IF bCalculateEnergySession THEN 
		//Socket 1
		IF FPMode3C2[1].Q OR FPMode3D2[1].Q THEN
			//Reset Counter when a new session is started
			stDataECSOut.arrSocketEnergySession[1] := 0;
				//Copy the Total Counter in kWh when a new session is started
				IF IsFinite(F_LREAL(arrSocketEnergySession[1])) THEN
					arrEnergySession_Cmp[1] := arrSocketEnergySession[1];
				END_IF
		END_IF
			IF (arrEnergySession_Cmp[1] <> arrSocketEnergySession[1] AND IsFinite(F_LREAL(arrSocketEnergySession[1])) AND (arrSocketMode3StateECS[1] = 'C2' OR arrSocketMode3StateECS[1] = 'D2')) THEN
				stDataECSOut.arrSocketEnergySession[1] := stDataECSOut.arrSocketEnergySession[1] + (arrSocketEnergySession[1] - arrEnergySession_Cmp[1]) / 1000;  
					stDataECSOut.arrSocketEnergySession[1] := stDataECSOut.arrSocketEnergySession[1];
						arrEnergySession_Cmp[1] := arrSocketEnergySession[1];		
			END_IF
		//Socket 2
		IF FPMode3C2[2].Q OR FPMode3D2[2].Q THEN
			//Reset Counter when a new session is started
			stDataECSOut.arrSocketEnergySession[2] := 0;
				//Copy the Total Counter in kWh when a new session is started
				IF IsFinite(F_LREAL(arrSocketEnergySession[2])) THEN
					arrEnergySession_Cmp[2] := arrSocketEnergySession[2];
				END_IF
		END_IF
			IF (arrEnergySession_Cmp[2] <> arrSocketEnergySession[2] AND IsFinite(F_LREAL(arrSocketEnergySession[2])) AND (arrSocketMode3StateECS[2] = 'C2' OR arrSocketMode3StateECS[2] = 'D2')) THEN
				stDataECSOut.arrSocketEnergySession[2] := stDataECSOut.arrSocketEnergySession[2] + (arrSocketEnergySession[2] - arrEnergySession_Cmp[2]) / 1000;  
					stDataECSOut.arrSocketEnergySession[2] := stDataECSOut.arrSocketEnergySession[2];
						arrEnergySession_Cmp[2] := arrSocketEnergySession[2];		
			END_IF
		//Socket 3
		IF FPMode3C2[3].Q OR FPMode3D2[3].Q THEN
			//Reset Counter when a new session is started
			stDataECSOut.arrSocketEnergySession[3] := 0;
				//Copy the Total Counter in kWh when a new session is started
				IF IsFinite(F_LREAL(arrSocketEnergySession[3])) THEN
					arrEnergySession_Cmp[3] := arrSocketEnergySession[3];
				END_IF
		END_IF
			IF (arrEnergySession_Cmp[3] <> arrSocketEnergySession[3] AND IsFinite(F_LREAL(arrSocketEnergySession[3])) AND (arrSocketMode3StateECS[3] = 'C2' OR arrSocketMode3StateECS[3] = 'D2')) THEN
				stDataECSOut.arrSocketEnergySession[3] := stDataECSOut.arrSocketEnergySession[3] + (arrSocketEnergySession[3] - arrEnergySession_Cmp[3]) / 1000;  
					stDataECSOut.arrSocketEnergySession[3] := stDataECSOut.arrSocketEnergySession[3];
						arrEnergySession_Cmp[3] := arrSocketEnergySession[3];		
			END_IF
		//Socket 4
		IF FPMode3C2[4].Q OR FPMode3D2[4].Q THEN
			//Reset Counter when a new session is started
			stDataECSOut.arrSocketEnergySession[4] := 0;
				//Copy the Total Counter in kWh when a new session is started
				IF IsFinite(F_LREAL(arrSocketEnergySession[4])) THEN
					arrEnergySession_Cmp[4] := arrSocketEnergySession[4];
				END_IF
		END_IF
			IF (arrEnergySession_Cmp[4] <> arrSocketEnergySession[4] AND IsFinite(F_LREAL(arrSocketEnergySession[4])) AND (arrSocketMode3StateECS[4] = 'C2' OR arrSocketMode3StateECS[4] = 'D2')) THEN
				stDataECSOut.arrSocketEnergySession[4] := stDataECSOut.arrSocketEnergySession[4] + (arrSocketEnergySession[4] - arrEnergySession_Cmp[4]) / 1000;  
					stDataECSOut.arrSocketEnergySession[4] := stDataECSOut.arrSocketEnergySession[4];
						arrEnergySession_Cmp[4] := arrSocketEnergySession[4];		
			END_IF
			
		stDataECSOut.arrSocketEnergySession[1] := LINT_TO_LREAL(LREAL_TO_LINT(stDataECSOut.arrSocketEnergySession[1] * 1000)) / 1000;
		stDataECSOut.arrSocketEnergySession[2] := LINT_TO_LREAL(LREAL_TO_LINT(stDataECSOut.arrSocketEnergySession[2] * 1000)) / 1000;
		stDataECSOut.arrSocketEnergySession[3] := LINT_TO_LREAL(LREAL_TO_LINT(stDataECSOut.arrSocketEnergySession[3] * 1000)) / 1000;
		stDataECSOut.arrSocketEnergySession[4] := LINT_TO_LREAL(LREAL_TO_LINT(stDataECSOut.arrSocketEnergySession[4] * 1000)) / 1000;
			
ELSE
	IF IsFinite(F_LREAL(arrSocketEnergySession[1])) THEN stDataECSOut.arrSocketEnergySession[1] := LINT_TO_LREAL(LREAL_TO_LINT((arrSocketEnergySession[1] / 1000) * 1000)) / 1000; END_IF
		IF IsFinite(F_LREAL(arrSocketEnergySession[2])) THEN stDataECSOut.arrSocketEnergySession[2] := LINT_TO_LREAL(LREAL_TO_LINT((arrSocketEnergySession[2] / 1000) * 1000)) / 1000; END_IF
			IF IsFinite(F_LREAL(arrSocketEnergySession[3])) THEN stDataECSOut.arrSocketEnergySession[3] := LINT_TO_LREAL(LREAL_TO_LINT((arrSocketEnergySession[3] / 1000) * 1000)) / 1000; END_IF
				IF IsFinite(F_LREAL(arrSocketEnergySession[4])) THEN stDataECSOut.arrSocketEnergySession[4] := LINT_TO_LREAL(LREAL_TO_LINT((arrSocketEnergySession[4] / 1000) * 1000)) / 1000; END_IF
END_IF
		
(*---------------------------------------------------------------------------Outputs--------------------------------------------------------------------------------------*)

stDataECSOut.byPriority := stSetupECS.byPriority;
	stDataECSOut.rMaxPower := DINT_TO_REAL(REAL_TO_DINT(stSetupECS.rMaxPower * 100)) / 100;
		stDataECSOut.bSOnEmergPowerOff := stSetupECS.bOnEmergPowerOff;
			stDataECSOut.bSManualyOn := stSetupECS.bManualyOn;
				stDataECSOut.bySManualyTargetPower := stSetupECS.byManualyTargetPower;
					stDataECSOut.bySCSMinPower := stSetupECS.byCSMinPower;

stDataECSOut.bCarConnected := bCarConnected;

//Mode 3 State
//Socket 1
//No Value.
IF arrSocketMode3StateECS[1] = '' OR arrSocketMode3StateECS[1] = 'F' OR NOT bEnable THEN
	stDataECSOut.arrSocketStateECS[1] := 0;
//ECS ready and Free	
ELSIF arrSocketMode3StateECS[1] = 'A' OR arrSocketMode3StateECS[1] = 'E' THEN
	stDataECSOut.arrSocketStateECS[1] := 1;
//Car Connected
ELSIF arrSocketMode3StateECS[1] = 'B1' OR arrSocketMode3StateECS[1] = 'B2' OR arrSocketMode3StateECS[1] = 'C1' OR arrSocketMode3StateECS[1] = 'D1' THEN
	stDataECSOut.arrSocketStateECS[1] := 2;
//Car Charging
ELSIF arrSocketMode3StateECS[1] = 'C2' OR arrSocketMode3StateECS[1] = 'D2' THEN
	stDataECSOut.arrSocketStateECS[1] := 3;
END_IF
//Socket 2
//No Value.
IF arrSocketMode3StateECS[2] = '' OR arrSocketMode3StateECS[2] = 'F' OR NOT bEnable THEN
	stDataECSOut.arrSocketStateECS[2] := 0;
//ECS ready and Free	
ELSIF arrSocketMode3StateECS[2] = 'A' OR arrSocketMode3StateECS[2] = 'E' THEN
	stDataECSOut.arrSocketStateECS[2] := 1;
//Car Connected
ELSIF arrSocketMode3StateECS[2] = 'B1' OR arrSocketMode3StateECS[2] = 'B2' OR arrSocketMode3StateECS[2] = 'C1' OR arrSocketMode3StateECS[2] = 'D1' THEN
	stDataECSOut.arrSocketStateECS[2] := 2;
//Car Charging
ELSIF arrSocketMode3StateECS[2] = 'C2' OR arrSocketMode3StateECS[2] = 'D2' THEN
	stDataECSOut.arrSocketStateECS[2] := 3;
END_IF
//Socket 3
//No Value.
IF arrSocketMode3StateECS[3] = '' OR arrSocketMode3StateECS[3] = 'F' OR NOT bEnable THEN
	stDataECSOut.arrSocketStateECS[3] := 0;
//ECS ready and Free	
ELSIF arrSocketMode3StateECS[3] = 'A' OR arrSocketMode3StateECS[3] = 'E' THEN
	stDataECSOut.arrSocketStateECS[3] := 1;
//Car Connected
ELSIF arrSocketMode3StateECS[3] = 'B1' OR arrSocketMode3StateECS[3] = 'B2' OR arrSocketMode3StateECS[3] = 'C1' OR arrSocketMode3StateECS[3] = 'D1' THEN
	stDataECSOut.arrSocketStateECS[3] := 2;
//Car Charging
ELSIF arrSocketMode3StateECS[3] = 'C2' OR arrSocketMode3StateECS[3] = 'D2' THEN
	stDataECSOut.arrSocketStateECS[3] := 3;
END_IF
//Socket 4
//No Value.
IF arrSocketMode3StateECS[4] = '' OR arrSocketMode3StateECS[4] = 'F' OR NOT bEnable THEN
	stDataECSOut.arrSocketStateECS[4] := 0;
//ECS ready and Free	
ELSIF arrSocketMode3StateECS[4] = 'A' OR arrSocketMode3StateECS[4] = 'E' THEN
	stDataECSOut.arrSocketStateECS[4] := 1;
//Car Connected
ELSIF arrSocketMode3StateECS[4] = 'B1' OR arrSocketMode3StateECS[4] = 'B2' OR arrSocketMode3StateECS[4] = 'C1' OR arrSocketMode3StateECS[4] = 'D1' THEN
	stDataECSOut.arrSocketStateECS[4] := 2;
//Car Charging
ELSIF arrSocketMode3StateECS[4] = 'C2' OR arrSocketMode3StateECS[4] = 'D2' THEN
	stDataECSOut.arrSocketStateECS[4] := 3;
END_IF
	
IF bEnable THEN
	stDataECSOut.arrSocketSOCCar[1] := arrSOCCar[1];
	stDataECSOut.arrSocketSOCCar[2] := arrSOCCar[2];
	stDataECSOut.arrSocketSOCCar[3] := arrSOCCar[3];
	stDataECSOut.arrSocketSOCCar[4] := arrSOCCar[4];
		stDataECSOut.arrChargingTimeInMin[1] := DINT_TO_REAL(REAL_TO_DINT(arrSocketChargingTimeInput[1] * 100)) / 100;
		stDataECSOut.arrChargingTimeInMin[2] := DINT_TO_REAL(REAL_TO_DINT(arrSocketChargingTimeInput[2] * 100)) / 100;
		stDataECSOut.arrChargingTimeInMin[3] := DINT_TO_REAL(REAL_TO_DINT(arrSocketChargingTimeInput[3] * 100)) / 100;
		stDataECSOut.arrChargingTimeInMin[4] := DINT_TO_REAL(REAL_TO_DINT(arrSocketChargingTimeInput[4] * 100)) / 100;
ELSE
	stDataECSOut.arrSocketSOCCar[1] := 0;
	stDataECSOut.arrSocketSOCCar[2] := 0;
	stDataECSOut.arrSocketSOCCar[3] := 0;
	stDataECSOut.arrSocketSOCCar[4] := 0;
		stDataECSOut.arrChargingTimeInMin[1] := 0;
		stDataECSOut.arrChargingTimeInMin[2] := 0;
		stDataECSOut.arrChargingTimeInMin[3] := 0;
		stDataECSOut.arrChargingTimeInMin[4] := 0;
END_IF

timDelayOutputs(IN:= bWriteWithDelay AND bEnable AND NOT timDelayOutputs.Q, PT:= tTimDelayOutput, Q=> , ET=> );
	FPEnable(CLK:= bEnable, Q=> );
		FNEnable(CLK:= bEnable, Q=> );
		
//Write with Delay or without
IF (bWriteWithDelay AND (timDelayOutputs.Q OR FPEnable.Q OR FNEnable.Q)) OR NOT bWriteWithDelay THEN
	stDataECSOutDelay := stDataECSOut;
END_IF

END_FUNCTION_BLOCK

// ---- Energy/FBs Internal/Electric Heating Element/FB_ElectricHeatingElement.TcPOU
{attribute 'conditionalshow'}
FUNCTION_BLOCK FB_ElectricHeatingElement
VAR_INPUT
	{attribute 'hide'}
	bEnable								: BOOL;									//Enable the Fuctionblock and his logic
	{attribute 'hide'}
	bError								: BOOL;									//Error Input electric heating element
	{attribute 'hide'}
	bWarning							: BOOL;									//Warning Input electric heating element
	{attribute 'hide'}
	bIsStepSwitched						: BOOL;									//Heating element is step switched or not
	{attribute 'hide'}
	bEPOIsActive						: BOOL;									//Emergency power operation is active
	{attribute 'hide'}
	bExternalLock						: BOOL;									//External lock (All functions are locked)
	{attribute 'hide'}
	bWriteWithDelay						: BOOL;									//Write with Delay the Data to the output (Not al Output Data is writen with Delay)
	{attribute 'hide'}
	bTimeDissableFunctions				: BOOL;									//True when we have longer Time no conncection to the Backend System. We need this Information to switch on the Heating Element for the Legionella Prtection
	{attribute 'hide'}
	iErrorCode							: INT;									//Error Code from external EHE
	{attribute 'hide'}
	iWarningCode						: INT;									//Warning Code from external EHE
	{attribute 'hide'}
	diNumberOfEHE						: DINT;									//Number of Electric Heating Element what is calculatet by a external function
	{attribute 'hide'}
	dwBatterySOC						: DWORD;								//Actual Battery SOC in %
	{attribute 'hide'}
	lrSizeGridConnection				: LREAL;								//Max size from the grid connection in kW
	{attribute 'hide'}
	lrGridPower							: LREAL;								//Actual Grid power in kW
	{attribute 'hide'}
	lrTotalCounterEnergy_Consumption	: LREAL;								//Total Counter for Energy consumption with unit Wh
	{attribute 'hide'}
	lrTotalCounterEnergy_Production		: LREAL;								//Total Counter for Energy production with unit Wh
	{attribute 'hide'}
	lrCounterEnergyT1_Consumption		: LREAL;								//Total counter for energy Tariff 1 consumption with unit Wh
	{attribute 'hide'}
	lrCounterEnergyT2_Consumption		: LREAL;								//Total counter for energy Tariff 2 consumption with unit Wh
	{attribute 'hide'}
	lrCounterEnergyT1_Production		: LREAL;								//Total counter for energy Tariff 1 production with unit Wh
	{attribute 'hide'}
	lrCounterEnergyT2_Production		: LREAL;								//Total counter for energy Tariff 2 production with unit Wh
	{attribute 'hide'}
	lrPowerEHE							: LREAL;								//Input Value from the power of the electro heating element with unit W
	{attribute 'hide'}
	arrTargetPower						: ARRAY[1..10] OF REAL;					//Target power from 0% to +100% for each step (0% to 100%) 
	{attribute 'hide'}
	rTemperatureInBoiler				: REAL;									//Temperature in the boiler which is heated with the heating element
	{attribute 'hide'}
	tTimDelayOutput						: TIME := T#5S;							//Delay Time to write some Data to the Output
	{attribute 'hide'}
	stSystemTime						: ST_Systemtime;						//Local System Time
	{attribute 'hide'}
	stSetupEHE							: ST_Setup_EHE;							//Setup electric heating element
END_VAR
VAR_OUTPUT
	{attribute 'hide'}
	stDataEHEOut						: ST_EHE_Output;						//Electric heating element output data
	{attribute 'hide'}
	stDataEHEOutDelay					: ST_EHE_Output;						//Electric heating element output data with delay
END_VAR
VAR
	{attribute 'hide'}
	fbPD1								: FB_PersistentData_Number;				//Function to save persistent data
	{attribute 'hide'}
	fbPD2								: FB_PersistentData_Number;				//Function to save persistent data
	{attribute 'hide'}
	FPTimeEnable						: R_TRIG;								//Internal positive edge
	{attribute 'hide'}
	FPTimeDisable						: R_TRIG;								//Internal positive edge
	{attribute 'hide'}
	FPWeekProgram						: R_TRIG;								//Internal positive edge
	{attribute 'hide'}
	FPRSWeekProgram						: R_TRIG;								//Internal positive edge
	{attribute 'hide'}
	FPEnable							: R_TRIG;								//Internal positive Edge
	{attribute 'hide'}
	FNEnable							: F_TRIG;								//Internal negative Edge
	{attribute 'hide'}
	timError							: TOF;									//Timer to set the error
	{attribute 'hide'}
	timWeekProgram						: TON;									//Timer for the week program (legionella protection)
	{attribute 'hide'}
	timDelayOutputs						: TON;									//Timer to send Data with Delay to the outputs
	{attribute 'hide'}
	timStep5							: TON;									//Timer what show when the state machine is to long in step 5. (The heating element not can heat the boiler at the Temperature what we need for the weekprogram)
	{attribute 'hide'}
	timStep6IsActive					: TON;									//Timer what is active when Step 6 in the State Machine is active
	{attribute 'hide'}
	timOnDelayStep6						: TON;									//Delay to switch on the EHE in Step 6
	{attribute 'hide'}
	timOffDelayStep6					: TON;									//Delay to switch off the EHE in Step 6
	{attribute 'hide'}
	timSOCOff							: TON;									//Timer to dissable the Device when the SOC from the Battery is under the Setpoint
	{attribute 'hide'}
	bTimeIsEnabled						: BOOL;									//Enable time controll
	{attribute 'hide'}
	byLPLimitsPw						: BYTE;									//Loop to check limits for target and max power
	{attribute 'hide'}
	byLPNumberOfSteps					: BYTE;									//Loop to ckeck to number of steps for step switching
	{attribute 'hide'}
	byLPMaxPowerOutput					: BYTE;									//Loop to ckeck the max power befor write to the output
	{attribute 'hide'}
	byLPSumPwOfSteps					: BYTE;									//Loop to calculate the complete power of all steps
	{attribute 'hide'}
	byLPPercentPwOfSteps				: BYTE;									//Loop to calculate the complete power in percent of all steps
	{attribute 'hide'}
	byLPMaxReached						: BYTE;									//Loop to check if for some step the target power is >= 100 or < Constants.byTargetOffPowerOnOffDevices
	{attribute 'hide'}
	iStateIntStep6						: INT;									//Internal Statmachine in Step 6
	{attribute 'hide'}
	uiState								: UINT;									//State Maschine
	{attribute 'hide'}
	uiHysteresisOnStep3					: UINT;									//Hysteresis to switch on or off the heating elemtn in step 3 (Surplus mode and max temperature)
	{attribute 'hide'}
	uiWeekProgramTemp					: UINT;									//Temperature, what is needed for the legionella protection
	{attribute 'hide'}
	rSumSteps							: REAL;									//Sum from all steps 
	{attribute 'hide'}
	arrMaxPower							: ARRAY[1..10] OF REAL; 				//Maximum power of the load in kW (Per stage) (If no stage or only On Off then max power in array[1])	
	{attribute 'hide'}
	arrPercentValueSteps				: ARRAY[1..10] OF REAL;					//Percent Value from each step
	{attribute 'hide'}
	arrMaxReached						: ARRAY[1..10] OF BOOL;					//Array from each step what goes to true when the power is >= 100%
END_VAR
VAR PERSISTENT
	{attribute 'conditionalshow'}
	bWeekProgramEnable					: BOOL;									//Enable the Week programm for one time
	{attribute 'conditionalshow'}
	byCounterDays						: BYTE;									//Counter that counts the days how long has not reached the maximum temperature
END_VAR

//Creator : Kai Ebensperger
//Company : Lynus AG
//Date : 19.05.2021
//Version : 1.0.0.0

//General description:
//This function block implements an electric heating element. It can be used for one adjustable step-switched, one adjustable stepless and one ON/OFF heating element.
//The function block can be switched manually and also contoll based.
//The output bOutputEHEOnOff is set at 100% power input. If the power input is < Constants.byTargetOffPowerOnOffDevices, the output is reset (hysteresis to prevent toggling).
//This output is used for electrical heating elements which cannot be controlled. So only have an on / off function. 
//The output bOutputEHE is set as soon as the power input is greater than or equal to 1%. This output is used for the control of the controllable heating elements. 
//If the temperature falls below the minimum temperature (uiTargetTempOn), the heating element is heated up until the target temperature (uiTargetTempOff) is reached. If time-controlled, this only takes place in the respectively enabled time.
//If a battery cabinet is in emergency power mode at this time, the current SOC must also be above the SOC Off value so that the heating element switches on. This prevents the battery from being discharged.
//IMPORTANT : When controlling the electric heating element, it is important that if it has an integrated mechanical thermostat, this value is set as high as the minimum max. temperature (uiTargetTempMax) set on the PLC. !!Min 65°C!!
//----------------------------------------
//Adjustable stage-switched heating element:
//With the controllable stage-switched heating element, each stage can be given a separate power setting. Each stage can be viewed internally similar to a heating element that can only ON/OFF.
//If >= 100% power output per stage, the percentage value of the respective stage is passed on to the power output (rTargetPowerEHE) or added to it. 
//If the level becomes < Constants.byTargetOffPowerOnOffDevices again, the percentage value is removed from the output again.
//----------------------------------------
//Adjustable stepless heating element:
//In the case of the controllable stepless heating element, the power setting is given linearly to the power setting output (rTargetPowerEHE). 
//The maximum power (arrMaxPowerEHE) must therefore only be entered in the first array field. 
//----------------------------------------
//On-off heating elemet
//Works in the same style like the stepless heating element. But here we use only the output bOutputEHEOnOff to switch on and off the heating element. The rTargetPowerEHE we didn't need here. 
//----------------------------------------
//Timefunctions: 
//If the time function has been selected, the heating element is only controlled if the uiTargetTempOn is undershot between the set time period.
//Is usefully if you have 2 differen current tariffs
//----------------------------------------
//Legionella protection: 
//If the Legionella protection has not been deactivated (bDisableLegionellaProtection), the heating element runs the maximum temperature once every 7 days (if the maximum temperature > 60°C), 
//or 60°C (if maximum temperature < 60°C). If within the 7 days the heating element has already reached the maximum temperature once, the counter, which counts the days will be reset.
//In emergency power mode, the program is only executed if the battery charge level allows it.
//When the Connection to the Backend is lost, then every 5 days the Heating Elemet switch on for 9 hours (In the 9 hours the temperature for legionella protection should be reached)
//----------------------------------------
//On Emergency power operation off
//If the lock for emergency power operation (bOnEmergPowerOff) has been selected for the electric heating element, it will not be switched on in emergency power operation. However, it can be overridden manually.
//----------------------------------------
//External look:
//The FB also has an external inhibit signal which switches off all functions as long as this signal is active.

(*---------------------------------------------------------------Check the limits of the inputs-------------------------------------------------------------------------------*)
dwBatterySOC := LIMIT(0, dwBatterySOC, 100);
	stSetupEHE.byManualyTargetPower := LIMIT(0, stSetupEHE.byManualyTargetPower, 100);
		rTemperatureInBoiler := LIMIT(-30, rTemperatureInBoiler, 120); 
			stSetupEHE.byHourOn := LIMIT(0, stSetupEHE.byHourOn, 23);
				stSetupEHE.byHourOff := LIMIT(0, stSetupEHE.byHourOff, 23);
					stSetupEHE.byMinutesOn := LIMIT(0, stSetupEHE.byMinutesOn, 59);
						stSetupEHE.byMinutesOff := LIMIT(0, stSetupEHE.byMinutesOff, 59);
						
IF IsFinite(F_LREAL(lrTotalCounterEnergy_Consumption)) THEN lrTotalCounterEnergy_Consumption := LIMIT(0,lrTotalCounterEnergy_Consumption,999999999999999); END_IF
	IF IsFinite(F_LREAL(lrTotalCounterEnergy_Production)) THEN lrTotalCounterEnergy_Production := LIMIT(0,lrTotalCounterEnergy_Production,999999999999999); END_IF
		IF IsFinite(F_LREAL(lrCounterEnergyT1_Consumption)) THEN lrCounterEnergyT1_Consumption := LIMIT(0,lrCounterEnergyT1_Consumption,999999999999999); END_IF
			IF IsFinite(F_LREAL(lrCounterEnergyT2_Consumption)) THEN lrCounterEnergyT2_Consumption := LIMIT(0,lrCounterEnergyT2_Consumption,999999999999999); END_IF
				IF IsFinite(F_LREAL(lrCounterEnergyT1_Production)) THEN lrCounterEnergyT1_Production := LIMIT(0,lrCounterEnergyT1_Production,999999999999999); END_IF
					IF IsFinite(F_LREAL(lrCounterEnergyT2_Production)) THEN lrCounterEnergyT2_Production := LIMIT(0,lrCounterEnergyT2_Production,999999999999999); END_IF
						lrPowerEHE := LIMIT(-999999999999999,lrPowerEHE,999999999999999);

//If a maximum power has not been entered everywhere, use the next higher power (only for step-switched). 
IF bIsStepSwitched AND stSetupEHE.rMaxPower1 <= 0 AND stSetupEHE.rMaxPower2 > 0 THEN 
	stSetupEHE.rMaxPower1 := stSetupEHE.rMaxPower2; 
END_IF
	IF bIsStepSwitched AND stSetupEHE.rMaxPower2 <= 0 AND stSetupEHE.rMaxPower3 > 0 THEN 
		stSetupEHE.rMaxPower2 := stSetupEHE.rMaxPower3;
	END_IF
IF bIsStepSwitched AND stSetupEHE.rMaxPower3 <= 0 AND stSetupEHE.rMaxPower4 > 0 THEN 
	stSetupEHE.rMaxPower3 := stSetupEHE.rMaxPower4; 
END_IF
	IF bIsStepSwitched AND stSetupEHE.rMaxPower4 <= 0 AND stSetupEHE.rMaxPower5 > 0 THEN 
		stSetupEHE.rMaxPower4 := stSetupEHE.rMaxPower5; 
	END_IF
IF bIsStepSwitched AND stSetupEHE.rMaxPower5 <= 0 AND stSetupEHE.rMaxPower6 > 0 THEN 
	stSetupEHE.rMaxPower5 := stSetupEHE.rMaxPower6; 
END_IF
	IF bIsStepSwitched AND stSetupEHE.rMaxPower6 <= 0 AND stSetupEHE.rMaxPower7 > 0 THEN 
		stSetupEHE.rMaxPower6 := stSetupEHE.rMaxPower7; 
	END_IF
IF bIsStepSwitched AND stSetupEHE.rMaxPower7 <= 0 AND stSetupEHE.rMaxPower8 > 0 THEN 
	stSetupEHE.rMaxPower7 := stSetupEHE.rMaxPower8; 
END_IF
	IF bIsStepSwitched AND stSetupEHE.rMaxPower8 <= 0 AND stSetupEHE.rMaxPower9 > 0 THEN 
		stSetupEHE.rMaxPower8 := stSetupEHE.rMaxPower9; 
	END_IF
IF bIsStepSwitched AND stSetupEHE.rMaxPower9 <= 0 AND stSetupEHE.rMaxPower10 > 0 THEN 
	stSetupEHE.rMaxPower9 := stSetupEHE.rMaxPower10; 
END_IF						

//Check limits for target power and maximum power						
FOR byLPLimitsPw := 1 TO 10 BY 1 DO
	arrTargetPower[byLPLimitsPw] := LIMIT(0, arrTargetPower[byLPLimitsPw], 100);
END_FOR
	stSetupEHE.rMaxPower1 := LIMIT(0,stSetupEHE.rMaxPower1,500);
		stSetupEHE.rMaxPower2 := LIMIT(0,stSetupEHE.rMaxPower2,500);
			stSetupEHE.rMaxPower3 := LIMIT(0,stSetupEHE.rMaxPower3,500);
				stSetupEHE.rMaxPower4 := LIMIT(0,stSetupEHE.rMaxPower4,500);
					stSetupEHE.rMaxPower5 := LIMIT(0,stSetupEHE.rMaxPower5,500);
						stSetupEHE.rMaxPower6 := LIMIT(0,stSetupEHE.rMaxPower6,500);
							stSetupEHE.rMaxPower7 := LIMIT(0,stSetupEHE.rMaxPower7,500);
								stSetupEHE.rMaxPower8 := LIMIT(0,stSetupEHE.rMaxPower8,500);
									stSetupEHE.rMaxPower9 := LIMIT(0,stSetupEHE.rMaxPower9,500);
										stSetupEHE.rMaxPower10 := LIMIT(0,stSetupEHE.rMaxPower10,500);

//Copy the max input power in the internal array to calculate the steps
arrMaxPower[1] := stSetupEHE.rMaxPower1;
	arrMaxPower[2] := stSetupEHE.rMaxPower2;
		arrMaxPower[3] := stSetupEHE.rMaxPower3;
			arrMaxPower[4] := stSetupEHE.rMaxPower4;
				arrMaxPower[5] := stSetupEHE.rMaxPower5;
					arrMaxPower[6] := stSetupEHE.rMaxPower6;
						arrMaxPower[7] := stSetupEHE.rMaxPower7;
							arrMaxPower[8] := stSetupEHE.rMaxPower8;
								arrMaxPower[9] := stSetupEHE.rMaxPower9;
									arrMaxPower[10] := stSetupEHE.rMaxPower10;

//Check that Disable SOC is bigger then Enable SOC	
IF stSetupEHE.byDisableSOC > stSetupEHE.byEnableSOC THEN 
	stSetupEHE.byEnableSOC := stSetupEHE.byDisableSOC + 1; 
END_IF
	stSetupEHE.byDisableSOC := LIMIT(0, stSetupEHE.byDisableSOC, 100);
		stSetupEHE.byEnableSOC := LIMIT(1, stSetupEHE.byEnableSOC, 100);

//Check that On temperature is bigger than off temperatur	
IF stSetupEHE.uiTargetTempOn > stSetupEHE.uiTargetTempOff THEN 
	stSetupEHE.uiTargetTempOff := stSetupEHE.uiTargetTempOn + 1; 
END_IF
	//Check that max temperature is bigger than on temperatur
	IF stSetupEHE.uiTargetTempOn > stSetupEHE.uiTargetTempMax THEN 
		stSetupEHE.uiTargetTempMax := stSetupEHE.uiTargetTempOn + 1; 
	END_IF
		//Check that max temperature is bigger than off temperatur
		IF stSetupEHE.uiTargetTempOff > stSetupEHE.uiTargetTempMax THEN 
			stSetupEHE.uiTargetTempMax := stSetupEHE.uiTargetTempOff + 1; 
		END_IF  
			stSetupEHE.uiTargetTempOn := LIMIT(0, stSetupEHE.uiTargetTempOn, 120);
				stSetupEHE.uiTargetTempOff := LIMIT(0, stSetupEHE.uiTargetTempOff, 120);
					stSetupEHE.uiTargetTempMax := LIMIT(0, stSetupEHE.uiTargetTempMax, 120);

//Calculate the hysteresis
IF stSetupEHE.uiTargetTempMax >= 2 THEN
	uiHysteresisOnStep3 := 1;
ELSE
	uiHysteresisOnStep3 := 0;
END_IF		

//Check number of steps
stDataEHEOut.byNumberOfSteps := 0;
	FOR byLPNumberOfSteps := 1 TO 10 BY 1 DO
		IF arrMaxPower[byLPNumberOfSteps] > 0 THEN stDataEHEOut.byNumberOfSteps := stDataEHEOut.byNumberOfSteps + 1; END_IF
	END_FOR

//Round the output power
FOR byLPMaxPowerOutput := 1 TO 10 BY 1 DO
	stDataEHEOut.arrMaxPower[byLPMaxPowerOutput] := DINT_TO_REAL(REAL_TO_DINT(arrMaxPower[byLPMaxPowerOutput] * 100)) / 100;
END_FOR	
		
(*---------------------------------------------------------------------------Enable----------------------------------------------------------------------------------*)
stDataEHEOut.bEnabled := bEnable;

(*-----------------------------------------------------------------------------Error and Warning----------------------------------------------------------------------------*)
timError(IN:= bError, PT:= T#5S, Q=> , ET=> );

stDataEHEOut.byErrorWarning := 0;
	IF bWarning OR timStep5.Q THEN stDataEHEOut.byErrorWarning := 1; END_IF 	
	IF timError.Q THEN stDataEHEOut.byErrorWarning := 2; END_IF

//Messages and Error Codes
IF stSetupEHE.bDisableLegionellaPr THEN stDataEHEOut.eMessage := E_Message_EHE.eLegionellaProtectionDisabledFromUser;
ELSIF timStep5.Q THEN stDataEHEOut.eMessage := E_Message_EHE.eEHEDontReachedTheSetTemp;
ELSIF bExternalLock THEN stDataEHEOut.eMessage := E_Message_EHE.eExternalLockActive;
ELSIF stDataEHEOut.byErrorWarning = 1 AND iWarningCode = 0 THEN stDataEHEOut.eMessage := E_Message_EHE.eNoConnectionToBackend;
ELSIF stDataEHEOut.byErrorWarning = 2 AND iErrorCode = 0 THEN stDataEHEOut.eMessage := E_Message_EHE.eErrorEHE;
ELSIF stDataEHEOut.byErrorWarning = 2 AND iErrorCode = 1 THEN stDataEHEOut.eMessage := E_Message_EHE.eTooMuchEHE;
ELSIF stDataEHEOut.byErrorWarning = 2 AND iErrorCode = 2 THEN stDataEHEOut.eMessage := E_Message_EHE.eTempSensorInBufferError;
ELSIF stDataEHEOut.byErrorWarning = 2 AND iErrorCode = 3 THEN stDataEHEOut.eMessage := E_Message_EHE.eWindowsSystemTimeError;	
ELSE stDataEHEOut.eMessage := E_Message_EHE.eNoMessage; 
END_IF
	
(*----------------------------------------------------------------------------Logic Part------------------------------------------------------------------------------------*)

//Timer for SOC dissabling
timSOCOff(IN:= dwBatterySOC <= stSetupEHE.byDisableSOC, PT:= T#30S, Q=> , ET=> );

//Switch heating element depending on temperature (without power setting, without control via time)
IF bEnable AND NOT bWeekProgramEnable AND NOT bExternalLock AND stDataEHEOut.byErrorWarning <> 2 AND 
 rTemperatureInBoiler < stSetupEHE.uiTargetTempOn AND NOT stSetupEHE.bTimeEnabled THEN 
	uiState := 1; 
END_IF

//Switch heating element depending on temperature (without power setting, with control via time)
IF bEnable AND NOT bWeekProgramEnable AND NOT bExternalLock AND stDataEHEOut.byErrorWarning <> 2 AND 
 rTemperatureInBoiler < stSetupEHE.uiTargetTempOn AND stSetupEHE.bTimeEnabled THEN 
	uiState := 2; 
END_IF

//Switch heating element with power preset (surplus)
IF bEnable AND NOT bWeekProgramEnable AND NOT bExternalLock AND stDataEHEOut.byErrorWarning <> 2 AND 
 (arrTargetPower[1] > 0 OR arrTargetPower[2] > 0 OR arrTargetPower[3] > 0 OR arrTargetPower[4] > 0 OR arrTargetPower[5] > 0 OR
 	arrTargetPower[6] > 0 OR arrTargetPower[7] > 0 OR arrTargetPower[8] > 0 OR arrTargetPower[9] > 0 OR arrTargetPower[10] > 0) THEN 
		uiState := 3; 
END_IF

//Switch heating element manually
IF bEnable AND NOT bWeekProgramEnable AND NOT bExternalLock AND stDataEHEOut.byErrorWarning <> 2 AND stSetupEHE.bManualyOn THEN 
	uiState := 4; 
END_IF 

//Legionella protection
IF NOT stSetupEHE.bDisableLegionellaPr THEN
	//Determine the temperature to be approached
	IF stSetupEHE.uiTargetTempMax > 60 THEN
		uiWeekProgramTemp := stSetupEHE.uiTargetTempMax;
	ELSE
		uiWeekProgramTemp := 60;
	END_IF
	
	//Timer and counter for days
	timWeekProgram(IN:= NOT timWeekProgram.Q AND bEnable AND uiState <> 5, PT:=T#24H , Q=> , ET=> );
		FPWeekProgram(CLK:= timWeekProgram.Q, Q=> );
			IF FPWeekProgram.Q THEN 
				byCounterDays := byCounterDays + 1; 
			END_IF
	
	//Reset the counter for the days
	FPRSWeekProgram(CLK:= rTemperatureInBoiler >= uiWeekProgramTemp, Q=> );		
		IF (byCounterDays >= 7 AND rTemperatureInBoiler >= uiWeekProgramTemp) OR FPRSWeekProgram.Q THEN 
			byCounterDays := 0; 
		END_IF
	
	IF byCounterDays >= 7 THEN 
		bWeekProgramEnable := TRUE;
	END_IF 
	
	IF bWeekProgramEnable THEN 
		uiState := 5; 
	END_IF
END_IF

//Timer, when the Weekprogram take to long time and dont reached the Week programm temperature
IF uiState = 5 THEN timStep5.IN := TRUE; ELSE timStep5.IN := FALSE; END_IF
	timStep5(IN:= , PT:= T#12H, Q=> , ET=> );

//Heating Element in Init step (Reset-Off)
IF NOT bEnable OR
	(uiState <> 5 AND (stDataEHEOut.byErrorWarning = 2 OR bExternalLock)) THEN
		uiState := 0;
END_IF

//Activeate the Legionella Protection when the Function is dissabled why we have no connection to the Backend Service
IF NOT bEnable AND bTimeDissableFunctions AND NOT stSetupEHE.bDisableLegionellaPr THEN uiState := 6; END_IF

//Enable via time
FPTimeEnable(CLK:= stSystemTime.wHour >= stSetupEHE.byHourOn AND stSystemTime.wMinute >= stSetupEHE.byMinutesOn AND stSetupEHE.bTimeEnabled, Q=> );
	FPTimeDisable(CLK:= stSystemTime.wHour >= stSetupEHE.byHourOff AND stSystemTime.wMinute >= stSetupEHE.byMinutesOff AND stSetupEHE.bTimeEnabled, Q=> );

IF FPTimeEnable.Q THEN 
	bTimeIsEnabled := TRUE; 
END_IF
	IF FPTimeDisable.Q THEN 
		bTimeIsEnabled := FALSE; 
	END_IF	
		IF NOT stSetupEHE.bTimeEnabled THEN 
			bTimeIsEnabled := FALSE; 
		END_IF

CASE uiState OF
	
	0: //Init step
		stDataEHEOut.bOutput := FALSE;
			stDataEHEOut.bOutputOnOff := FALSE;
				stDataEHEOut.rTargetPower := 0;
			
	1: //Switch heating element depending on temperature (without power setting, without control via time)
		IF (rTemperatureInBoiler < stSetupEHE.uiTargetTempOn AND NOT bEPOIsActive) OR (rTemperatureInBoiler < stSetupEHE.uiTargetTempOn AND 
		 bEPOIsActive AND NOT stSetupEHE.bOnEmergPowerOff AND dwBatterySOC >= stSetupEHE.byEnableSOC)	THEN 
			stDataEHEOut.bOutput := TRUE; 
				stDataEHEOut.bOutputOnOff := TRUE; 
					stDataEHEOut.rTargetPower := 100;
		END_IF
		
		IF (rTemperatureInBoiler >= stSetupEHE.uiTargetTempOff) OR (timSOCOff.Q AND bEPOIsActive) OR 
		 (bEPOIsActive AND stSetupEHE.bOnEmergPowerOff) THEN
			stDataEHEOut.bOutput := FALSE; 
				stDataEHEOut.bOutputOnOff := FALSE; 
					stDataEHEOut.rTargetPower := 0;
		END_IF
		 
	2: //Switch heating element depending on temperature (without power setting, with control via time)	
		IF (rTemperatureInBoiler < stSetupEHE.uiTargetTempOn AND NOT bEPOIsActive AND bTimeIsEnabled) OR 
			(rTemperatureInBoiler < stSetupEHE.uiTargetTempOn AND bEPOIsActive AND NOT stSetupEHE.bOnEmergPowerOff AND dwBatterySOC >= stSetupEHE.byEnableSOC AND bTimeIsEnabled) THEN 
				stDataEHEOut.bOutput := TRUE; stDataEHEOut.bOutputOnOff := TRUE; stDataEHEOut.rTargetPower := 100; 
		END_IF
			IF (rTemperatureInBoiler >= stSetupEHE.uiTargetTempOff) OR 
				(timSOCOff.Q AND bEPOIsActive) OR
					(bEPOIsActive AND stSetupEHE.bOnEmergPowerOff) OR	 
						NOT bTimeIsEnabled THEN
							stDataEHEOut.bOutput := FALSE; stDataEHEOut.bOutputOnOff := FALSE; stDataEHEOut.rTargetPower := 0;
			END_IF

	3: //Switch heating element with power preset (surplus)
		//Power not stepped switched (on-off or linear)
		IF NOT bIsStepSwitched AND stDataEHEOut.byNumberOfSteps > 0 THEN	
			stDataEHEOut.rTargetPower := DINT_TO_REAL(REAL_TO_DINT(arrTargetPower[1] * 100)) / 100;
		END_IF
		
		//Power step switched
		//Calculate the sum of power from al steps
		rSumSteps := 0;
		FOR byLPSumPwOfSteps := 1 TO 10 BY 1 DO
			rSumSteps := rSumSteps + stDataEHEOut.arrMaxPower[byLPSumPwOfSteps];
				arrPercentValueSteps[byLPSumPwOfSteps] := 0;	
		END_FOR
		
		//Calculate the power in % for each step	
		IF stDataEHEOut.byNumberOfSteps > 0 AND stDataEHEOut.byNumberOfSteps <= 10 AND rSumSteps > 0 THEN
			FOR byLPPercentPwOfSteps := 1 TO stDataEHEOut.byNumberOfSteps BY 1 DO
				arrPercentValueSteps[byLPPercentPwOfSteps] := (stDataEHEOut.arrMaxPower[byLPPercentPwOfSteps] * 100) / rSumSteps;
			END_FOR 
		END_IF
		
		//Check when a step has reached the maximum or not	
		FOR byLPMaxReached := 1 TO 10 BY 1 DO
			IF arrTargetPower[byLPMaxReached] >= 100 THEN 
				arrMaxReached[byLPMaxReached] := TRUE; 
			END_IF	
				IF arrTargetPower[byLPMaxReached] < Constants_Energy.byTargetOffPowerForOnOffDevices THEN 
					arrMaxReached[byLPMaxReached] := FALSE; 
				END_IF	
		END_FOR
		
		//Off	
		IF bIsStepSwitched AND stDataEHEOut.byNumberOfSteps > 0 AND NOT arrMaxReached[1] AND arrTargetPower[1] < Constants_Energy.byTargetOffPowerForOnOffDevices THEN 
			stDataEHEOut.rTargetPower := 0; 
		END_IF 
		//Step 1
		IF bIsStepSwitched AND stDataEHEOut.byNumberOfSteps > 0 AND arrMaxReached[1] AND arrTargetPower[1] >= Constants_Energy.byTargetOffPowerForOnOffDevices THEN 
			stDataEHEOut.rTargetPower := DINT_TO_REAL(REAL_TO_DINT(arrPercentValueSteps[1] * 100)) / 100; 	
		END_IF
		//Step 1 to Step 2
		IF bIsStepSwitched AND stDataEHEOut.byNumberOfSteps > 0 AND arrMaxReached[1] AND arrMaxReached[2] AND arrTargetPower[2] >= Constants_Energy.byTargetOffPowerForOnOffDevices THEN 
			stDataEHEOut.rTargetPower := DINT_TO_REAL(REAL_TO_DINT((arrPercentValueSteps[1] + arrPercentValueSteps[2]) * 100)) / 100; 
		END_IF
		//Step 1 to Step 3
		IF bIsStepSwitched AND stDataEHEOut.byNumberOfSteps > 0 AND arrMaxReached[1] AND arrMaxReached[2] AND arrMaxReached[3] AND 
		 arrTargetPower[3] >= Constants_Energy.byTargetOffPowerForOnOffDevices THEN 
			stDataEHEOut.rTargetPower := DINT_TO_REAL(REAL_TO_DINT((arrPercentValueSteps[1] + arrPercentValueSteps[2] + arrPercentValueSteps[3]) * 100)) / 100; 
		END_IF
		//Step 1 to Step 4				
		IF bIsStepSwitched AND stDataEHEOut.byNumberOfSteps > 0 AND arrMaxReached[1] AND arrMaxReached[2] AND arrMaxReached[3] AND 
		 arrMaxReached[4] AND arrTargetPower[4] >= Constants_Energy.byTargetOffPowerForOnOffDevices THEN 
			stDataEHEOut.rTargetPower := DINT_TO_REAL(REAL_TO_DINT((arrPercentValueSteps[1] + arrPercentValueSteps[2] + 
				arrPercentValueSteps[3] + arrPercentValueSteps[4]) * 100)) / 100; 
		END_IF
		//Step 1 to Step 5					
		IF bIsStepSwitched AND stDataEHEOut.byNumberOfSteps > 0 AND arrMaxReached[1] AND arrMaxReached[2] AND arrMaxReached[3] AND
		 arrMaxReached[4] AND arrMaxReached[5] AND arrTargetPower[5] >= Constants_Energy.byTargetOffPowerForOnOffDevices THEN 
			stDataEHEOut.rTargetPower := DINT_TO_REAL(REAL_TO_DINT((arrPercentValueSteps[1] + arrPercentValueSteps[2] + 
				arrPercentValueSteps[3] + arrPercentValueSteps[4] + arrPercentValueSteps[5]) * 100)) / 100; 
		END_IF
		//Step 1 to Step 6
		IF bIsStepSwitched AND stDataEHEOut.byNumberOfSteps > 0 AND arrMaxReached[1] AND arrMaxReached[2] AND arrMaxReached[3] AND 
		 arrMaxReached[4] AND arrMaxReached[5] AND arrMaxReached[6] AND arrTargetPower[6] >= Constants_Energy.byTargetOffPowerForOnOffDevices THEN 
			stDataEHEOut.rTargetPower := DINT_TO_REAL(REAL_TO_DINT((arrPercentValueSteps[1] + arrPercentValueSteps[2] + 
				arrPercentValueSteps[3] + arrPercentValueSteps[4] + arrPercentValueSteps[5] + arrPercentValueSteps[6]) * 100)) / 100; 
		END_IF
		//Step 1 to Step 7	
		IF bIsStepSwitched AND stDataEHEOut.byNumberOfSteps > 0 AND arrMaxReached[1] AND arrMaxReached[2] AND arrMaxReached[3] AND 
		 arrMaxReached[4] AND arrMaxReached[5] AND arrMaxReached[6] AND arrMaxReached[7] AND arrTargetPower[7] >= Constants_Energy.byTargetOffPowerForOnOffDevices THEN 
			stDataEHEOut.rTargetPower := DINT_TO_REAL(REAL_TO_DINT((arrPercentValueSteps[1] + arrPercentValueSteps[2] + 
				arrPercentValueSteps[3] + arrPercentValueSteps[4] + arrPercentValueSteps[5] + arrPercentValueSteps[6] + arrPercentValueSteps[7]) * 100)) / 100; 
		END_IF
		//Step 1 to Step 8
		IF bIsStepSwitched AND stDataEHEOut.byNumberOfSteps > 0 AND arrMaxReached[1] AND arrMaxReached[2] AND arrMaxReached[3] AND 
		 arrMaxReached[4] AND arrMaxReached[5] AND arrMaxReached[6] AND arrMaxReached[7] AND arrMaxReached[8] AND arrTargetPower[8] >= Constants_Energy.byTargetOffPowerForOnOffDevices THEN 
			stDataEHEOut.rTargetPower := DINT_TO_REAL(REAL_TO_DINT((arrPercentValueSteps[1] + arrPercentValueSteps[2] + 
				arrPercentValueSteps[3] + arrPercentValueSteps[4] + arrPercentValueSteps[5] + arrPercentValueSteps[6] + arrPercentValueSteps[7] + 
					arrPercentValueSteps[8]) * 100)) / 100; 
		END_IF
		//Step 1 to Step 9
		IF bIsStepSwitched AND stDataEHEOut.byNumberOfSteps > 0 AND arrMaxReached[1] AND arrMaxReached[2] AND arrMaxReached[3] AND 
		 arrMaxReached[4] AND arrMaxReached[5] AND arrMaxReached[6] AND arrMaxReached[7] AND arrMaxReached[8] AND arrMaxReached[9] AND arrTargetPower[9] >= Constants_Energy.byTargetOffPowerForOnOffDevices THEN 
			stDataEHEOut.rTargetPower := DINT_TO_REAL(REAL_TO_DINT((arrPercentValueSteps[1] + arrPercentValueSteps[2] + 
				arrPercentValueSteps[3] + arrPercentValueSteps[4] + arrPercentValueSteps[5] + arrPercentValueSteps[6] + arrPercentValueSteps[7] + 
					arrPercentValueSteps[8] + arrPercentValueSteps[9]) * 100)) / 100; 
		END_IF
		//Step 1 to Step 10
		IF bIsStepSwitched AND stDataEHEOut.byNumberOfSteps > 0 AND arrMaxReached[1] AND arrMaxReached[2] AND arrMaxReached[3] AND 
		 arrMaxReached[4] AND arrMaxReached[5] AND arrMaxReached[6] AND arrMaxReached[7] AND arrMaxReached[8] AND arrMaxReached[9] AND arrMaxReached[10] AND 
			 arrTargetPower[10] >= Constants_Energy.byTargetOffPowerForOnOffDevices THEN 
				stDataEHEOut.rTargetPower := DINT_TO_REAL(REAL_TO_DINT((arrPercentValueSteps[1] + arrPercentValueSteps[2] + 
					arrPercentValueSteps[3] + arrPercentValueSteps[4] + arrPercentValueSteps[5] + arrPercentValueSteps[6] + arrPercentValueSteps[7] + 
						arrPercentValueSteps[8] + arrPercentValueSteps[9] + arrPercentValueSteps[10]) * 100)) / 100; 
		END_IF
		//Limit the output to <= 100
		IF bIsStepSwitched AND stDataEHEOut.rTargetPower > 100 THEN 
			stDataEHEOut.rTargetPower := 100; 
		END_IF 
			
		//Swtich the outputs
		IF (NOT bEPOIsActive AND (arrTargetPower[1] > 0 OR arrTargetPower[2] > 0 OR arrTargetPower[3] > 0 OR arrTargetPower[4] > 0 OR arrTargetPower[5] > 0 OR
		 arrTargetPower[6] > 0 OR arrTargetPower[7] > 0 OR arrTargetPower[8] > 0 OR arrTargetPower[9] > 0 OR arrTargetPower[10] > 0) AND
		 dwBatterySOC >= stSetupEHE.byEnableSOC AND rTemperatureInBoiler < stSetupEHE.uiTargetTempMax - uiHysteresisOnStep3) OR 
		 (bEPOIsActive AND NOT stSetupEHE.bOnEmergPowerOff AND (arrTargetPower[1] > 0 OR arrTargetPower[2] > 0 OR arrTargetPower[3] > 0 OR 
		 arrTargetPower[4] > 0 OR arrTargetPower[5] > 0 OR arrTargetPower[6] > 0 OR arrTargetPower[7] > 0 OR arrTargetPower[8] > 0 OR 
		 arrTargetPower[9] > 0 OR arrTargetPower[10] > 0) AND dwBatterySOC >= stSetupEHE.byEnableSOC AND 
		 rTemperatureInBoiler < stSetupEHE.uiTargetTempMax - uiHysteresisOnStep3) THEN
			stDataEHEOut.bOutput := TRUE;
		END_IF
		
		IF (arrTargetPower[1] <= 0 AND arrTargetPower[2] <= 0 AND arrTargetPower[3] <= 0 AND arrTargetPower[4] <= 0 AND arrTargetPower[5] <= 0 AND
		 arrTargetPower[6] <= 0 AND arrTargetPower[7] <= 0 AND arrTargetPower[8] <= 0 AND arrTargetPower[9] <= 0 AND arrTargetPower[10] <= 0) OR 
		 timSOCOff.Q OR (bEPOIsActive AND stSetupEHE.bOnEmergPowerOff) OR rTemperatureInBoiler >= stSetupEHE.uiTargetTempMax OR
		 stDataEHEOut.byNumberOfSteps <= 0 THEN
			stDataEHEOut.bOutput := FALSE;
		END_IF 	
		
		IF NOT stDataEHEOut.bOutput THEN 
			stDataEHEOut.rTargetPower := 0; 
		END_IF 
			IF stDataEHEOut.rTargetPower >= 100 AND stDataEHEOut.bOutput THEN 
				stDataEHEOut.bOutputOnOff := TRUE; 
			END_IF
				IF stDataEHEOut.rTargetPower < Constants_Energy.byTargetOffPowerForOnOffDevices OR NOT stDataEHEOut.bOutput THEN 
					stDataEHEOut.bOutputOnOff := FALSE; 
				END_IF 

	4: //Switch heating element manually
		stDataEHEOut.rTargetPower := BYTE_TO_REAL(stSetupEHE.byManualyTargetPower);
		
		IF stSetupEHE.bManualyOn AND stDataEHEOut.rTargetPower > 0 THEN 
			stDataEHEOut.bOutput := TRUE; 
		END_IF
			IF NOT stSetupEHE.bManualyOn OR stDataEHEOut.rTargetPower <= 0 THEN 
				stDataEHEOut.bOutput := FALSE; 
			END_IF 
				IF NOT stDataEHEOut.bOutput THEN 
					stDataEHEOut.rTargetPower := 0; 
				END_IF 	
					IF stDataEHEOut.rTargetPower >= 100 AND stDataEHEOut.bOutput THEN 
						stDataEHEOut.bOutputOnOff := TRUE; 
					END_IF
						IF stDataEHEOut.rTargetPower < Constants_Energy.byTargetOffPowerForOnOffDevices OR NOT stDataEHEOut.bOutput THEN 
							stDataEHEOut.bOutputOnOff := FALSE; 
						END_IF	
	
	5: //Week programm (Legionella protection)
		//100% target power
		IF (bEPOIsActive AND dwBatterySOC >= stSetupEHE.byEnableSOC AND bWeekProgramEnable AND stDataEHEOut.byErrorWarning <> 2 AND NOT bExternalLock) OR (NOT bEPOIsActive AND bWeekProgramEnable AND stDataEHEOut.byErrorWarning <> 2 AND NOT bExternalLock) THEN 
			stDataEHEOut.bOutput := TRUE; 
				stDataEHEOut.bOutputOnOff := TRUE; 
					stDataEHEOut.rTargetPower := 100;
		END_IF
			//Off when emergency power operation is on and battery soc is to low	
			IF (bEPOIsActive AND timSOCOff.Q) OR stDataEHEOut.byErrorWarning = 2 OR bExternalLock THEN
				stDataEHEOut.bOutput := FALSE; 
					stDataEHEOut.bOutputOnOff := FALSE; 
						stDataEHEOut.rTargetPower := 0;
			END_IF
				//Finish and back to the init step
				IF FPRSWeekProgram.Q OR stSetupEHE.bDisableLegionellaPr THEN 
					bWeekProgramEnable := FALSE; 
						uiState := 0; 
				END_IF
				
	6://Legionelle Protection when we have no connection to the Backend Service
		
		CASE iStateIntStep6 OF

			0://Init Step
				timStep6IsActive.IN := TRUE;
					IF timStep6IsActive.Q THEN iStateIntStep6 := 1; timStep6IsActive.IN := FALSE; END_IF
			
			1://Wait that we have enought Power on the Grid
				IF (lrGridPower + stSetupEHE.rMaxPower1 + stSetupEHE.rMaxPower2 + stSetupEHE.rMaxPower3 + stSetupEHE.rMaxPower4 + stSetupEHE.rMaxPower5 + 
						stSetupEHE.rMaxPower6 + stSetupEHE.rMaxPower7 + stSetupEHE.rMaxPower8 + stSetupEHE.rMaxPower9 + stSetupEHE.rMaxPower10) <= lrSizeGridConnection AND diNumberOfEHE > 0 THEN
					timOnDelayStep6.IN := TRUE;
				ELSE
					timOnDelayStep6.IN := FALSE;
				END_IF  	
					//Next Step
					IF timOnDelayStep6.Q THEN iStateIntStep6 := 2; timOnDelayStep6.IN := FALSE; END_IF
					
			2://Switch on the Electric Heating Elemnt with the Max Power for 9 hours
				stDataEHEOut.rTargetPower := 100;
					stDataEHEOut.bOutput := TRUE;
						stDataEHEOut.bOutputOnOff := TRUE;
							timOffDelayStep6.IN := TRUE;	
					//Next Step
					IF timOffDelayStep6.Q THEN 
						iStateIntStep6 := 0; 
							stDataEHEOut.bOutput := FALSE;
								stDataEHEOut.bOutputOnOff := FALSE;
									stDataEHEOut.rTargetPower := 0; 
										timOffDelayStep6.IN := FALSE;
					END_IF
				
		END_CASE 
	
		//End of this Step
		IF NOT bTimeDissableFunctions OR bEnable OR stSetupEHE.bDisableLegionellaPr THEN uiState := 0; iStateIntStep6 := 0; END_IF  
	
END_CASE

//Timer for Step 6 (Legionella protection when we have no connerction to the Backend Service)
IF uiState <> 6 THEN 
	timStep6IsActive.IN := FALSE; 
		timOnDelayStep6.IN := FALSE; 
			timOffDelayStep6.IN := FALSE;
END_IF
			
timStep6IsActive(IN:= , PT:= T#5D, Q=> , ET=> );
	timOnDelayStep6(IN:= , PT:= (T#1M * diNumberOfEHE), Q=> , ET=> );
		timOffDelayStep6(IN:= , PT:= T#9H, Q=> , ET=> );

(*------------------------------------------------------------------Power data----------------------------------------------------------------------------------------------*)
IF bEnable THEN	
	stDataEHEOut.lrPower := LINT_TO_LREAL(LREAL_TO_LINT((lrPowerEHE / 1000) * 100)) / 100;
		IF IsFinite(F_LREAL(lrCounterEnergyT1_Consumption)) THEN stDataEHEOut.lrCounterEnergyT1_Consumption := LINT_TO_LREAL(LREAL_TO_LINT((lrCounterEnergyT1_Consumption / 1000) * 100)) / 100; END_IF
			IF IsFinite(F_LREAL(lrCounterEnergyT2_Consumption)) THEN stDataEHEOut.lrCounterEnergyT2_Consumption := LINT_TO_LREAL(LREAL_TO_LINT((lrCounterEnergyT2_Consumption / 1000) * 100)) / 100; END_IF
				IF IsFinite(F_LREAL(lrCounterEnergyT1_Production)) THEN stDataEHEOut.lrCounterEnergyT1_Production := LINT_TO_LREAL(LREAL_TO_LINT((lrCounterEnergyT1_Production / 1000) * 100)) / 100; END_IF
					IF IsFinite(F_LREAL(lrCounterEnergyT2_Production)) THEN stDataEHEOut.lrCounterEnergyT2_Production := LINT_TO_LREAL(LREAL_TO_LINT((lrCounterEnergyT2_Production / 1000) * 100)) / 100; END_IF
						IF IsFinite(F_LREAL(lrTotalCounterEnergy_Consumption)) THEN stDataEHEOut.lrTotalCounterEnergy_Consumption := LINT_TO_LREAL(LREAL_TO_LINT((lrTotalCounterEnergy_Consumption / 1000) * 100)) / 100; END_IF
							IF IsFinite(F_LREAL(lrTotalCounterEnergy_Production)) THEN stDataEHEOut.lrTotalCounterEnergy_Production := LINT_TO_LREAL(LREAL_TO_LINT((lrTotalCounterEnergy_Production / 1000) * 100)) / 100; END_IF 	
			
	IF stDataEHEOut.lrPower < 0 THEN
		stDataEHEOut.lrPowerProduction := (stDataEHEOut.lrPower * - 1);
		stDataEHEOut.lrPowerConsumption := 0;
	ELSIF stDataEHEOut.lrPower > 0 THEN
		stDataEHEOut.lrPowerProduction := 0;
		stDataEHEOut.lrPowerConsumption := stDataEHEOut.lrPower;
	ELSIF stDataEHEOut.lrPower = 0 THEN
		stDataEHEOut.lrPowerProduction := 0;
		stDataEHEOut.lrPowerConsumption := 0;
	END_IF
		
ELSE
	stDataEHEOut.lrPower := 0;
		stDataEHEOut.lrCounterEnergyT1_Consumption := 0;
			stDataEHEOut.lrCounterEnergyT2_Consumption := 0;
				stDataEHEOut.lrCounterEnergyT1_Production := 0;
					stDataEHEOut.lrCounterEnergyT2_Production := 0;
						stDataEHEOut.lrPowerProduction := 0;
							stDataEHEOut.lrPowerConsumption := 0;	
								stDataEHEOut.lrTotalCounterEnergy_Consumption := 0;
									stDataEHEOut.lrTotalCounterEnergy_Production := 0;
END_IF

(*---------------------------------------------------------------------------Outputs--------------------------------------------------------------------------------------*)
stDataEHEOut.byPriority := stSetupEHE.byPriority;
	stDataEHEOut.bIsStepSwitched := bIsStepSwitched;
		stDataEHEOut.bSOnEmergPowerOff := stSetupEHE.bOnEmergPowerOff;
			stDataEHEOut.bSManualyOn := stSetupEHE.bManualyOn;
				stDataEHEOut.bySManualyTargetPower := stSetupEHE.byManualyTargetPower;
					stDataEHEOut.bSTimeEnabled := stSetupEHE.bTimeEnabled;
						stDataEHEOut.bSDisableLegionellaPr := stSetupEHE.bDisableLegionellaPr;
					
IF bEnable THEN
	stDataEHEOut.rTempInBoiler := DINT_TO_REAL(REAL_TO_DINT(rTemperatureInBoiler * 100)) / 100;
ELSE	
	stDataEHEOut.rTempInBoiler := 0;
END_IF

timDelayOutputs(IN:= bWriteWithDelay AND bEnable AND NOT timDelayOutputs.Q, PT:= tTimDelayOutput, Q=> , ET=> );
	FPEnable(CLK:= bEnable, Q=> );
		FNEnable(CLK:= bEnable, Q=> );

//Write with Delay or without
IF (bWriteWithDelay AND (timDelayOutputs.Q OR FPEnable.Q OR FNEnable.Q)) OR NOT bWriteWithDelay THEN
	stDataEHEOutDelay := stDataEHEOut;
END_IF
		
(*----------------------------------------------------------Save persistent data----------------------------------------------------------------*)
fbPD1(lrValue:= BOOL_TO_REAL(bWeekProgramEnable), bEventBasedActive=> );
	fbPD2(lrValue:= BYTE_TO_REAL(byCounterDays), bEventBasedActive=> );

END_FUNCTION_BLOCK

// ---- Persistent Data/FBs Internal/PD Slave/FB_PersistentData_Number.TcPOU
{attribute 'hide_all_locals'}
{attribute 'conditionalshow'}
FUNCTION_BLOCK FB_PersistentData_Number
VAR_INPUT
	{attribute 'hide'}
	lrValue								: LREAL;				//Actual Input Value
END_VAR
VAR_OUTPUT
	{attribute 'hide'}
	bEventBasedActive					: BOOL;					//Event based saving is active
END_VAR
VAR
	lrValue_CP							: LREAL;				//Value to compare the input Value
	fbTaskIndex							: GETCURTASKINDEX;		//Get the Task index
END_VAR

//Creator : Kai Ebensperger
//Company : Lynus AG
//Date : 15.02.2021
//Version : 1.0.0.0

//With this Function we can check if the Value on the Input of the Function ha changed an chan start to saving the persistent Data in Event Based Mode
//Work only with Number Fromat

//---------------------------------------------------------------Logic to start the save process---------------------------------------------------------------------------------------

bEventBasedActive := GVL_Persistent_Data.bEventBasedActive;

//After Restart the System set the Variables direct to actual value because they are loadet from the card
fbTaskIndex(index=> );
	IF TwinCAT_SystemInfoVarList._TaskInfo[fbTaskIndex.index].FirstCycle THEN lrValue_CP := lrValue; END_IF

IF NOT GVL_Persistent_Data.bBusy AND bEventBasedActive AND lrValue <> lrValue_CP THEN
	GVL_Persistent_Data.bSaveData := TRUE;
		lrValue_CP := lrValue;
END_IF

END_FUNCTION_BLOCK

// ---- Energy/FBs Internal/Electric Meter/FB_ElectricMeter.TcPOU
{attribute 'hide_all_locals'}
{attribute 'conditionalshow'}
FUNCTION_BLOCK FB_ElectricMeter
VAR_INPUT
	{attribute 'hide'}
	bEnable								: BOOL;											//Enable the function
	{attribute 'hide'}
	bError								: BOOL;											//Error from the meter
	{attribute 'hide'}
	bWarning							: BOOL;											//Warning from the meter
	{attribute 'hide'}
	bEnableReadOutFunction				: BOOL;											//Enable the output to Read out the Meter
	{attribute 'hide'}
	bWriteWithDelay						: BOOL;											//Write with Delay the Data to the output (Not al Output Data is writen with Delay)
	{attribute 'hide'}
	bPowerDataInvers					: BOOL;											//With True its possible to invert all received power data from the electric meter
	{attribute 'hide'}
	bReadOutDataDone					: BOOL;											//With this Input you can send the command to the Function that the reading out from the data is done
	{attribute 'hide'}
	iTimeReadOutInterval				: INT;											//Delay in seconds to read out the electric meter
	{attribute 'hide'}
	iErrorCode							: INT;											//Error Code from external EHE
	{attribute 'hide'}
	iWarningCode						: INT;											//Warning Code from external EHE
	{attribute 'hide'}
	lrTotalCounterEnergy_Consumption	: LREAL;										//Total Counter for Energy consumption with unit kWh
	{attribute 'hide'}
	lrTotalCounterEnergy_Production		: LREAL;										//Total Counter for Energy production with unit kWh
	{attribute 'hide'}
	lrCounterEnergyT1_Consumption		: LREAL;										//Total counter for energy Tariff 1 consumption with unit kWh
	{attribute 'hide'}
	lrCounterEnergyT2_Consumption		: LREAL;										//Total counter for energy Tariff 2 consumption with unit kWh
	{attribute 'hide'}
	lrCounterEnergyT1_Production		: LREAL;										//Total counter for energy Tariff 1 production with unit kWh
	{attribute 'hide'}
	lrCounterEnergyT2_Production		: LREAL;										//Total counter for energy Tariff 2 production with unit kWh
	{attribute 'hide'}
	lrCurrentL1							: LREAL;										//Current from L1 with unit A
	{attribute 'hide'}
	lrVoltageL1N						: LREAL;										//Voltage L1-N with unit V
	{attribute 'hide'}
	lrVoltageL1L2						: LREAL;										//Voltage L1-L2 with unit V
	{attribute 'hide'}
	lrPowerL1							: LREAL;										//Power L1 with unit W
	{attribute 'hide'}
	lrCurrentL2							: LREAL;										//Current from L2 with unit A
	{attribute 'hide'}
	lrVoltageL2N						: LREAL;										//Voltage L2-N with unit V
	{attribute 'hide'}
	lrVoltageL2L3						: LREAL;										//Voltage L2-L3 with unit V
	{attribute 'hide'}
	lrPowerL2							: LREAL;										//Power L2 with unit W
	{attribute 'hide'}
	lrCurrentL3							: LREAL;										//Current from L3 with unit A
	{attribute 'hide'}
	lrVoltageL3N						: LREAL;										//Voltage L3-N with unit V
	{attribute 'hide'}
	lrVoltageL3L1						: LREAL;										//Voltage L3-L1 with unit V
	{attribute 'hide'}
	lrPowerL3							: LREAL;										//Power L3 with unit W
	{attribute 'hide'}
	lrPowerTotal						: LREAL;										//Total power with unit W
	{attribute 'hide'}		
	lrFrequency							: LREAL;										//Frequency with unit HZ
	{attribute 'hide'}
	lrReactivePowerTotal				: LREAL;										//Reactive power with unit var
	{attribute 'hide'}
	lrApparentPowerTotal				: LREAL;										//Apparent Power with unit VA
	{attribute 'hide'}
	tTimDelayOutput						: TIME := T#5S;									//Delay Time to write some Data to the Output
END_VAR                             	
VAR_OUTPUT    
	{attribute 'hide'}                      	
	stDataEMOutPower					: ST_ElectricMeter_Output_Power;				//Electric meter power output data
	{attribute 'hide'}
	stDataEMOutPowerDelay				: ST_ElectricMeter_Output_Power;				//Electric meter power output data with delay
	{attribute 'hide'}
	bReadOutMeter						: BOOL;											//Pulse to read out the meter
END_VAR 
VAR_OUTPUT PERSISTENT
	{attribute 'conditionalshow'}                     	
	stDataEMOutCounter					: ST_ElectricMeter_Output_Counter;				//Electric meter counter output data
	{attribute 'conditionalshow'}
	stDataEMOutCounterDelay				: ST_ElectricMeter_Output_Counter;				//Electric meter counter output data with delay
END_VAR                            	
VAR       
	FPEnable							: R_TRIG;										//Internal positive edge
	FNEnable							: F_TRIG;										//Internal negative Edge  
	FNReadOutDone						: F_TRIG;                        				//Internal negative Edge 
	tim0								: TON;											//Timer for read out time
	tim1								: TON;											//Timer reset read out
	timDelayOutputs						: TON;											//Timer to send Data with Delay to the outputs
	timSavePD							: TON;											//Timer to save the persistent Data when the Event Based Mode is active
	arrPD								: ARRAY[1..12] OF FB_PersistentData_Number;		//Function to save persistent data
END_VAR

//Creator : Kai Ebensperger
//Company : Lynus AG
//Date : 20.05.2021
//Version : 1.0.0.0

//With this function block can read in data from a electric couter.
//The time how often the meter is reading out can be selected on the inputs
//The Counter Values are saved persistend only every 6 hours when the Event Based Mode is active on the Persistend Master Function Block

(*---------------------------------------------------------------Check the limits of the inputs-------------------------------------------------------------------------------*)
iTimeReadOutInterval := LIMIT(1,iTimeReadOutInterval,3600);

IF IsFinite(F_LREAL(lrTotalCounterEnergy_Consumption)) THEN lrTotalCounterEnergy_Consumption := LIMIT(0,lrTotalCounterEnergy_Consumption,999999999999999); END_IF
	IF IsFinite(F_LREAL(lrTotalCounterEnergy_Production)) THEN lrTotalCounterEnergy_Production := LIMIT(0,lrTotalCounterEnergy_Production,999999999999999); END_IF
		IF IsFinite(F_LREAL(lrCounterEnergyT1_Consumption)) THEN lrCounterEnergyT1_Consumption := LIMIT(0,lrCounterEnergyT1_Consumption,999999999999999); END_IF
			IF IsFinite(F_LREAL(lrCounterEnergyT2_Consumption)) THEN lrCounterEnergyT2_Consumption := LIMIT(0,lrCounterEnergyT2_Consumption,999999999999999); END_IF
				IF IsFinite(F_LREAL(lrCounterEnergyT1_Production)) THEN lrCounterEnergyT1_Production := LIMIT(0,lrCounterEnergyT1_Production,999999999999999); END_IF
					IF IsFinite(F_LREAL(lrCounterEnergyT2_Production)) THEN lrCounterEnergyT2_Production := LIMIT(0,lrCounterEnergyT2_Production,999999999999999); END_IF

lrPowerL1 := LIMIT(-999999999999999,lrPowerL1,999999999999999);
	lrPowerL2 := LIMIT(-999999999999999,lrPowerL2,999999999999999);	
		lrPowerL3 := LIMIT(-999999999999999,lrPowerL3,999999999999999);	
			lrPowerTotal := LIMIT(-999999999999999,lrPowerTotal,999999999999999);	
			
lrReactivePowerTotal := LIMIT(-999999999999999,lrReactivePowerTotal,999999999999999);
	lrApparentPowerTotal := LIMIT(-999999999999999,lrApparentPowerTotal,999999999999999);	
	
lrCurrentL1 := LIMIT(-999999999999999,lrCurrentL1,999999999999999);
	lrCurrentL2 := LIMIT(-999999999999999,lrCurrentL2,999999999999999);
		lrCurrentL3 := LIMIT(-999999999999999,lrCurrentL3,999999999999999);

lrVoltageL1N := LIMIT(0,lrVoltageL1N,100000);
	lrVoltageL1L2 := LIMIT(0,lrVoltageL1L2,100000);
lrVoltageL2N := LIMIT(0,lrVoltageL2N,100000);
	lrVoltageL2L3 := LIMIT(0,lrVoltageL2L3,100000);
lrVoltageL3N := LIMIT(0,lrVoltageL3N,100000);
	lrVoltageL3L1 := LIMIT(0,lrVoltageL3L1,100000);

lrFrequency := LIMIT(0,lrFrequency,200);

(*------------------------------------------------------------------------------------Activate to read out the meter-------------------------------------------------------------------*)
FPEnable(CLK:= bEnable, Q=> );

tim0(IN:= NOT tim0.Q, PT:= (T#1S * iTimeReadOutInterval) , Q=> , ET=> );
	IF (bEnableReadOutFunction AND (tim0.Q OR FPEnable.Q)) THEN
		bReadOutMeter := TRUE;
	END_IF
	
tim1(IN:= bReadOutMeter, PT:=T#100MS , Q=> , ET=> );
	IF tim1.Q OR NOT bEnableReadOutFunction THEN
		bReadOutMeter := FALSE;
	END_IF		

(*------------------------------------------------------------------------------------Error and Warning-----------------------------------------------------------------------*)	

stDataEMOutPower.byErrorWarning := 0;
	IF bWarning THEN stDataEMOutPower.byErrorWarning := 1; END_IF  
	IF bError THEN stDataEMOutPower.byErrorWarning := 2; END_IF

//Messages and Error Codes
IF stDataEMOutPower.byErrorWarning = 1 AND iWarningCode = 0 THEN stDataEMOutPower.eMessage := E_Message_EM.eNoConnectionToBackend;
ELSIF stDataEMOutPower.byErrorWarning = 1 AND iWarningCode = 1 THEN stDataEMOutPower.eMessage := E_Message_EM.eElectricMeterWarning;
ELSIF stDataEMOutPower.byErrorWarning = 2 AND iErrorCode = 0 THEN stDataEMOutPower.eMessage := E_Message_EM.eElectricMeterError;
ELSIF stDataEMOutPower.byErrorWarning = 2 AND iErrorCode = 1 THEN stDataEMOutPower.eMessage := E_Message_EM.eTooMuchElectricMeter;
ELSE stDataEMOutPower.eMessage := E_Message_EM.eNoMessage; 
END_IF
	
(*-------------------------------------------------------------------------------------------Data from the meter----------------------------------------------------------------------------*)

timDelayOutputs(IN:= bWriteWithDelay AND bEnable AND NOT timDelayOutputs.Q, PT:= tTimDelayOutput, Q=> , ET=> );
	FPEnable(CLK:= bEnable, Q=> );
			FNEnable(CLK:= bEnable, Q=> );	

//Counter Data
FNReadOutDone(CLK:= bReadOutDataDone, Q=> );

IF FNReadOutDone.Q AND NOT bError THEN
	IF IsFinite(F_LREAL(lrTotalCounterEnergy_Production)) THEN stDataEMOutCounter.lrTotalCounterEnergy_Production := LINT_TO_LREAL(LREAL_TO_LINT(lrTotalCounterEnergy_Production * 100)) / 100; END_IF
	IF IsFinite(F_LREAL(lrTotalCounterEnergy_Consumption)) THEN stDataEMOutCounter.lrTotalCounterEnergy_Consumption := LINT_TO_LREAL(LREAL_TO_LINT(lrTotalCounterEnergy_Consumption * 100)) / 100; END_IF
	IF IsFinite(F_LREAL(lrCounterEnergyT1_Consumption)) THEN stDataEMOutCounter.lrCounterEnergyT1_Consumption := LINT_TO_LREAL(LREAL_TO_LINT(lrCounterEnergyT1_Consumption * 100)) / 100; END_IF
	IF IsFinite(F_LREAL(lrCounterEnergyT2_Consumption)) THEN stDataEMOutCounter.lrCounterEnergyT2_Consumption := LINT_TO_LREAL(LREAL_TO_LINT(lrCounterEnergyT2_Consumption * 100)) / 100; END_IF
	IF IsFinite(F_LREAL(lrCounterEnergyT1_Production)) THEN stDataEMOutCounter.lrCounterEnergyT1_Production := LINT_TO_LREAL(LREAL_TO_LINT(lrCounterEnergyT1_Production * 100)) / 100; END_IF
	IF IsFinite(F_LREAL(lrCounterEnergyT2_Production)) THEN stDataEMOutCounter.lrCounterEnergyT2_Production := LINT_TO_LREAL(LREAL_TO_LINT(lrCounterEnergyT2_Production * 100)) / 100; END_IF
END_IF		
			
//Power Data
IF bEnable THEN
	stDataEMOutPower.lrPowerTotal := lrPowerTotal / 1000;
	stDataEMOutPower.lrPowerTotal := LINT_TO_LREAL(LREAL_TO_LINT(stDataEMOutPower.lrPowerTotal * 100)) / 100;
	IF NOT bPowerDataInvers THEN
		IF 	stDataEMOutPower.lrPowerTotal < 0 THEN
			stDataEMOutPower.lrPowerProduction := (stDataEMOutPower.lrPowerTotal * - 1);
			stDataEMOutPower.lrPowerConsumption := 0;
		ELSIF stDataEMOutPower.lrPowerTotal > 0 THEN
			stDataEMOutPower.lrPowerProduction := 0;
			stDataEMOutPower.lrPowerConsumption := stDataEMOutPower.lrPowerTotal;
		ELSIF stDataEMOutPower.lrPowerTotal = 0 THEN
			stDataEMOutPower.lrPowerProduction := 0;
			stDataEMOutPower.lrPowerConsumption := 0;
		END_IF
	ELSE
		IF 	stDataEMOutPower.lrPowerTotal < 0 THEN
			stDataEMOutPower.lrPowerProduction := 0;
			stDataEMOutPower.lrPowerConsumption := (stDataEMOutPower.lrPowerTotal * - 1);
		ELSIF stDataEMOutPower.lrPowerTotal > 0 THEN
			stDataEMOutPower.lrPowerProduction := stDataEMOutPower.lrPowerTotal;
			stDataEMOutPower.lrPowerConsumption := 0;
		ELSIF stDataEMOutPower.lrPowerTotal = 0 THEN
			stDataEMOutPower.lrPowerProduction := 0;
			stDataEMOutPower.lrPowerConsumption := 0;
		END_IF
	END_IF										
	stDataEMOutPower.lrReactivePowerTotal := lrReactivePowerTotal / 1000;
	stDataEMOutPower.lrReactivePowerTotal := LINT_TO_LREAL(LREAL_TO_LINT(stDataEMOutPower.lrReactivePowerTotal * 100)) / 100;
	stDataEMOutPower.lrApparentPowerTotal := lrApparentPowerTotal / 1000;
	stDataEMOutPower.lrApparentPowerTotal := LINT_TO_LREAL(LREAL_TO_LINT(stDataEMOutPower.lrApparentPowerTotal * 100)) / 100;											
	stDataEMOutPower.lrFrequency := LINT_TO_LREAL(LREAL_TO_LINT(lrFrequency * 100)) / 100;;
	stDataEMOutPower.lrVoltageL1N := LINT_TO_LREAL(LREAL_TO_LINT(lrVoltageL1N * 100)) / 100;
	stDataEMOutPower.lrVoltageL1L2 := LINT_TO_LREAL(LREAL_TO_LINT(lrVoltageL1L2 * 100)) / 100;
	stDataEMOutPower.lrCurrentL1 := LINT_TO_LREAL(LREAL_TO_LINT(lrCurrentL1 * 100)) / 100;
	stDataEMOutPower.lrPowerL1 :=  lrPowerL1 / 1000;
	stDataEMOutPower.lrPowerL1 := LINT_TO_LREAL(LREAL_TO_LINT(stDataEMOutPower.lrPowerL1 * 100)) / 100;
	stDataEMOutPower.lrVoltageL2N := LINT_TO_LREAL(LREAL_TO_LINT(lrVoltageL2N * 100)) / 100;
	stDataEMOutPower.lrVoltageL2L3 := LINT_TO_LREAL(LREAL_TO_LINT(lrVoltageL2L3 * 100)) / 100;
	stDataEMOutPower.lrCurrentL2 := LINT_TO_LREAL(LREAL_TO_LINT(lrCurrentL2 * 100)) / 100;
	stDataEMOutPower.lrPowerL2 := lrPowerL2 / 1000;
	stDataEMOutPower.lrPowerL2 := LINT_TO_LREAL(LREAL_TO_LINT(stDataEMOutPower.lrPowerL2 * 100)) / 100;
	stDataEMOutPower.lrVoltageL3N := LINT_TO_LREAL(LREAL_TO_LINT(lrVoltageL3N * 100)) / 100;
	stDataEMOutPower.lrVoltageL3L1 := LINT_TO_LREAL(LREAL_TO_LINT(lrVoltageL3L1 * 100)) / 100;
	stDataEMOutPower.lrCurrentL3 := LINT_TO_LREAL(LREAL_TO_LINT(lrCurrentL3 * 100)) / 100;
	stDataEMOutPower.lrPowerL3 := lrPowerL3 / 1000;
	stDataEMOutPower.lrPowerL3 := LINT_TO_LREAL(LREAL_TO_LINT(stDataEMOutPower.lrPowerL3 * 100)) / 100;
		stDataEMOutPower.bEnabled := bEnable;	
ELSE																																														
	stDataEMOutPower.lrPowerTotal := 0;
	stDataEMOutPower.lrPowerProduction := 0;
	stDataEMOutPower.lrPowerConsumption := 0;
	stDataEMOutPower.lrReactivePowerTotal := 0;
	stDataEMOutPower.lrApparentPowerTotal := 0;
	stDataEMOutPower.lrFrequency := 0;
	stDataEMOutPower.lrVoltageL1N := 0;
	stDataEMOutPower.lrVoltageL1L2 := 0;
	stDataEMOutPower.lrCurrentL1 := 0;
	stDataEMOutPower.lrPowerL1 := 0;
	stDataEMOutPower.lrVoltageL2N := 0;
	stDataEMOutPower.lrVoltageL2L3 := 0;
	stDataEMOutPower.lrCurrentL2 := 0;
	stDataEMOutPower.lrPowerL2 := 0;
	stDataEMOutPower.lrVoltageL3N := 0;
	stDataEMOutPower.lrVoltageL3L1 := 0;
	stDataEMOutPower.lrCurrentL3 := 0;
	stDataEMOutPower.lrPowerL3 := 0;
		stDataEMOutPower.bEnabled := bEnable;
	
	bReadOutMeter := FALSE;																							
END_IF			

(*---------------------------------------------------------------Outputs-------------------------------------------------------------------------------*)

//Write with Delay or without
IF (bWriteWithDelay AND (timDelayOutputs.Q OR FPEnable.Q OR FNEnable.Q)) OR NOT bWriteWithDelay THEN
	stDataEMOutPowerDelay := stDataEMOutPower; 
		stDataEMOutCounterDelay := stDataEMOutCounter;
END_IF 

(*----------------------------------------------------------Save persistent data----------------------------------------------------------------*)

//When the Event Based mode is active, save the Data only every 6h
//When we have this Function Blocks in the plc code use the Mode "Power Fail" if the PLC System has this possibility
timSavePD(IN:= GVL_Persistent_Data.bEventBasedActive AND NOT timSavePD.Q, PT:= T#6H, Q=> , ET=> );

IF timSavePD.Q THEN
	arrPD[1].lrValue := stDataEMOutCounter.lrCounterEnergyT1_Consumption;
	arrPD[2].lrValue := stDataEMOutCounter.lrCounterEnergyT1_Production;
	arrPD[3].lrValue := stDataEMOutCounter.lrCounterEnergyT2_Consumption; 
	arrPD[4].lrValue := stDataEMOutCounter.lrCounterEnergyT2_Production;
	arrPD[5].lrValue := stDataEMOutCounter.lrTotalCounterEnergy_Consumption;
	arrPD[6].lrValue := stDataEMOutCounter.lrTotalCounterEnergy_Production;
	arrPD[7].lrValue := stDataEMOutCounterDelay.lrCounterEnergyT1_Consumption;
	arrPD[8].lrValue := stDataEMOutCounterDelay.lrCounterEnergyT1_Production;
	arrPD[9].lrValue := stDataEMOutCounterDelay.lrCounterEnergyT2_Consumption;
	arrPD[10].lrValue := stDataEMOutCounterDelay.lrCounterEnergyT2_Production;
	arrPD[11].lrValue := stDataEMOutCounterDelay.lrTotalCounterEnergy_Consumption;
	arrPD[12].lrValue := stDataEMOutCounterDelay.lrTotalCounterEnergy_Production;
END_IF

arrPD[1](lrValue:= , bEventBasedActive=> );
arrPD[2](lrValue:= , bEventBasedActive=> );
arrPD[3](lrValue:= , bEventBasedActive=> );
arrPD[4](lrValue:= , bEventBasedActive=> );
arrPD[5](lrValue:= , bEventBasedActive=> );
arrPD[6](lrValue:= , bEventBasedActive=> );
arrPD[7](lrValue:= , bEventBasedActive=> );
arrPD[8](lrValue:= , bEventBasedActive=> );
arrPD[9](lrValue:= , bEventBasedActive=> );
arrPD[10](lrValue:= , bEventBasedActive=> );
arrPD[11](lrValue:= , bEventBasedActive=> );
arrPD[12](lrValue:= , bEventBasedActive=> );

END_FUNCTION_BLOCK

// ---- Energy/FBs Internal/EMS/FB_EMS_Message.TcPOU
{attribute 'conditionalshow'}
FUNCTION_BLOCK FB_EMS_Message
VAR_INPUT
	{attribute 'hide'}
	bEnable									: BOOL;								//Enable/Dissable the Function
	{attribute 'hide'}
	wMessageCode							: WORD;								//External Message Code
END_VAR
VAR_OUTPUT
	{attribute 'hide'}
	eMessageEMS								: E_Message_EMS;					//EMS Message
END_VAR
VAR
END_VAR

//Creator : Kai Ebensperger
//Company : Lynus AG
//Date : 10.05.21
//Version : 1.0.0.0

//With this Function its possible to create messages for the EMS function on the plc

IF bEnable AND wMessageCode = 0 THEN eMessageEMS := E_Message_EMS.eEnabled; END_IF
IF bEnable AND wMessageCode = 1 THEN eMessageEMS := E_Message_EMS.eAllPrioritysAtMinimum; END_IF
IF bEnable AND wMessageCode = 2 THEN eMessageEMS := E_Message_EMS.eAllPrioritysAtMaximum; END_IF
IF bEnable AND wMessageCode = 3 THEN eMessageEMS := E_Message_EMS.eMissingPowerValuesOnDeviceSetup; END_IF
IF bEnable AND wMessageCode = 4 THEN eMessageEMS := E_Message_EMS.eTooMuchFunctionsInThisProject; END_IF
IF bEnable AND wMessageCode = 5 THEN eMessageEMS := E_Message_EMS.eNoConnectionToBackend; END_IF

IF NOT bEnable THEN eMessageEMS := E_Message_EMS.eDisabled; END_IF

END_FUNCTION_BLOCK

// ---- Energy/FBs Internal/Energy Counter/FB_EnergyCounter.TcPOU
{attribute 'hide_all_locals'}
{attribute 'conditionalshow'}
FUNCTION_BLOCK FB_EnergyCounter
VAR_INPUT
	{attribute 'hide'}
	byActiveTariff						: BYTE;													//Active Tariff
	{attribute 'hide'}
	lrPowerInput						: LREAL;												//Input Power in kW
END_VAR
VAR_OUTPUT PERSISTENT
	{attribute 'conditionalshow'}
	lrTotalCounterEnergy_Consumption	: LREAL;												//Total Counter for Energy consumption with unit kWh
	{attribute 'conditionalshow'}
	lrTotalCounterEnergy_Production		: LREAL;												//Total Counter for Energy production with unit kWh
	{attribute 'conditionalshow'}
	lrCounterEnergyT1_Consumption		: LREAL;												//Total counter for energy Tariff 1 consumption with unit kWh
	{attribute 'conditionalshow'}	
	lrCounterEnergyT2_Consumption		: LREAL;												//Total counter for energy Tariff 2 consumption with unit kWh
	{attribute 'conditionalshow'}
	lrCounterEnergyT1_Production		: LREAL;												//Total counter for energy Tariff 1 production with unit kWh
	{attribute 'conditionalshow'}
	lrCounterEnergyT2_Production		: LREAL;												//Total counter for energy Tariff 2 production with unit kWh
END_VAR
VAR
	arrPD								: ARRAY[1..6] OF FB_PersistentData_Number;				//Function to save persistent data
	timSavePD							: TON;													//Timer to save the persistent Data when the Event Based Mode is active
	timNewValue							: TON;													//Timer to copy every second a new power value
	TaskInfo							: GETCURTASKINDEX;										//Function to get the Task Index
	byWorkMode							: BYTE;													//Work Mode for calculation (1 = Production, 2 = Consumption)
	udiCycleTime						: UDINT;												//Cycle Time
	lrCyclesForSecond					: LREAL;												//Needed cycles for 1 Second
	uiCounterConsumption				: UINT;													//Counter for Cycles in Consumption Mode
	uiSecondsConsumption				: UINT;													//Elapses Seconds for Consumption
	rHourConsumption					: REAL;													//Elapsed Hours for Consumption
	uiCounterProduction					: UINT;													//Counter for Cycles in Production Mode
	uiSecondsProduction					: UINT;													//Elapses Seconds for Production
	rHourProduction						: REAL;													//Elapsed Hours for Production
	lrPowerInput_Int					: LREAL;												//Input Power in kW
	lrkW_Consumption_CP					: LREAL;												//Power to compare in Consumption Mode
	lrkW_Production_CP					: LREAL;												//Powet to compare in Production Mode
END_VAR

//Creator : Kai Ebensperger
//Company : Lynus AG
//Date : 16.11.2021
//Version : 1.0.0.0

//This function block can be used to count different Energy Counter
//Positive Values mens comsumption
//Negative Values means production 

(*--------------------------------------------------------------------------Limits-----------------------------------------------------------------------------------*)

byActiveTariff := LIMIT(1,byActiveTariff,2);

(*---------------------------------------------------------------------------Logic-----------------------------------------------------------------------------------*)

//Get Task Index
TaskInfo(index=> );
	//Cycle Time in ms
	IF TwinCAT_SystemInfoVarList._TaskInfo[TaskInfo.index].CycleTime <> 0 THEN
		udiCycleTime := TwinCAT_SystemInfoVarList._TaskInfo[TaskInfo.index].CycleTime / 10000;
	END_IF

//Cycles for 1 Second
IF udiCycleTime > 0 THEN 
	lrCyclesForSecond := (1 / UDINT_TO_LREAL(udiCycleTime)) * 1000; 
END_IF

//Timer to copy the new Value
//Necessary becaue the rest of the logic can handly min every second a change on the power side
timNewValue(IN:= NOT timNewValue.Q, PT:= T#1S, Q=> , ET=> );
	IF timNewValue.Q THEN lrPowerInput_Int := lrPowerInput; END_IF

IF lrCyclesForSecond <> 0 THEN

	uiCounterConsumption := uiCounterConsumption + 1;
		uiCounterProduction := uiCounterProduction + 1;
	
	//Calculate the Time	
	IF uiCounterProduction >= lrCyclesForSecond THEN uiSecondsProduction := uiSecondsProduction + 1; uiCounterProduction := 0; END_IF
		rHourProduction := UINT_TO_REAL(uiSecondsProduction) / 3600;
	IF uiCounterConsumption >= lrCyclesForSecond THEN uiSecondsConsumption := uiSecondsConsumption + 1; uiCounterConsumption := 0; END_IF
		rHourConsumption := UINT_TO_REAL(uiSecondsConsumption) / 3600;
	
	//Production
	IF lrkW_Production_CP <> lrPowerInput_Int THEN
		IF byWorkMode = 1 THEN 
			//Production Tariff 1
			IF byActiveTariff = 1 THEN 
				lrCounterEnergyT1_Production := lrCounterEnergyT1_Production + ((lrkW_Production_CP * - 1) * rHourProduction); 
					lrkW_Production_CP := lrPowerInput_Int;
			END_IF
			//Production Tariff 2
			IF byActiveTariff = 2 THEN 
				lrCounterEnergyT2_Production := lrCounterEnergyT2_Production + ((lrkW_Production_CP * - 1) * rHourProduction); 
					lrkW_Production_CP := lrPowerInput_Int;
			END_IF
		ELSE
			lrkW_Production_CP := 0;
		END_IF
				rHourProduction := 0; uiSecondsProduction := 0;  uiCounterProduction := 0;	
	END_IF
	
	//Consumption
	IF lrkW_Consumption_CP <> lrPowerInput_Int THEN
		IF byWorkMode = 2 THEN  
			//Consumption Tariff 1
			IF byActiveTariff = 1 THEN 
				lrCounterEnergyT1_Consumption := lrCounterEnergyT1_Consumption + (lrkW_Consumption_CP * rHourConsumption); 
					lrkW_Consumption_CP := lrPowerInput_Int;
			END_IF
			//Consumption Tariff 2
			IF byActiveTariff = 2 THEN 
				lrCounterEnergyT2_Consumption := lrCounterEnergyT2_Consumption + (lrkW_Consumption_CP * rHourConsumption); 
					lrkW_Consumption_CP := lrPowerInput_Int;
			END_IF
		ELSE
			lrkW_Consumption_CP := 0;
		END_IF
				rHourConsumption := 0; uiSecondsConsumption := 0;  uiCounterConsumption := 0;	
	END_IF

END_IF

//Total Consumption and Production
lrTotalCounterEnergy_Consumption := lrCounterEnergyT1_Consumption + lrCounterEnergyT2_Consumption;
	lrTotalCounterEnergy_Production := lrCounterEnergyT1_Production + lrCounterEnergyT2_Production;

//Switch between the Work modes
IF lrPowerInput_Int <= 0 THEN byWorkMode := 1; ELSE byWorkMode := 2; END_IF 
	
(*----------------------------------------------------------Save persistent data----------------------------------------------------------------*)

//When the Event Based mode is active, save the Data only every 6h
//When we have this Function Blocks in the plc code use the Mode "Power Fail" if the PLC System has this possibility
timSavePD(IN:= GVL_Persistent_Data.bEventBasedActive AND NOT timSavePD.Q, PT:= T#6H, Q=> , ET=> );

IF timSavePD.Q THEN
	arrPD[1].lrValue := lrTotalCounterEnergy_Consumption;
	arrPD[2].lrValue := lrTotalCounterEnergy_Production;
	arrPD[3].lrValue := lrCounterEnergyT1_Consumption; 
	arrPD[4].lrValue := lrCounterEnergyT2_Consumption;
	arrPD[5].lrValue := lrCounterEnergyT1_Production;
	arrPD[6].lrValue := lrCounterEnergyT2_Production;
END_IF

arrPD[1](lrValue:= , bEventBasedActive=> );
arrPD[2](lrValue:= , bEventBasedActive=> );
arrPD[3](lrValue:= , bEventBasedActive=> );
arrPD[4](lrValue:= , bEventBasedActive=> );
arrPD[5](lrValue:= , bEventBasedActive=> );
arrPD[6](lrValue:= , bEventBasedActive=> );

END_FUNCTION_BLOCK

// ---- Energy/FBs Internal/Generator/FB_Generator.TcPOU
{attribute 'hide_all_locals'}
{attribute 'conditionalshow'}
FUNCTION_BLOCK FB_Generator
VAR_INPUT
	{attribute 'hide'}
	bEnable								: BOOL;									//Enable or disable this function
	{attribute 'hide'}
	bError								: BOOL;									//Generator has a error
	{attribute 'hide'}
	bWarning							: BOOL;									//Generator has a warning
	{attribute 'hide'}
	bReset								: BOOL;									//Reset the function after a error (Read the Reset output back with a negative edge because send a active reset signal to the generator)
	{attribute 'hide'}
	bWriteWithDelay						: BOOL;									//Write with Delay the Data to the output (Not al Output Data is writen with Delay)
	{attribute 'hide'}
	iErrorCode							: INT;									//Error Code from external Generator
	{attribute 'hide'}
	iWarningCode						: INT;									//Warning Code from external Generator
	{attribute 'hide'}
	dwBatterySOC						: DWORD;								//Actual Battery SOC in %
	{attribute 'hide'}
	lrTotalCounterEnergy_Consumption	: LREAL;								//Total Counter for Energy consumption with unit Wh
	{attribute 'hide'}
	lrTotalCounterEnergy_Production		: LREAL;								//Total Counter for Energy production with unit Wh
	{attribute 'hide'}
	lrCounterEnergyT1_Consumption		: LREAL;								//Total counter for energy Tariff 1 consumption with unit Wh
	{attribute 'hide'}
	lrCounterEnergyT2_Consumption		: LREAL;								//Total counter for energy Tariff 2 consumption with unit Wh
	{attribute 'hide'}
	lrCounterEnergyT1_Production		: LREAL;								//Total counter for energy Tariff 1 production with unit Wh
	{attribute 'hide'}
	lrCounterEnergyT2_Production		: LREAL;								//Total counter for energy Tariff 2 production with unit Wh
	{attribute 'hide'}
	lrPowerGenerator					: LREAL;								//Input Value from the power of the Generator with unit W
	{attribute 'hide'}
	tDelaySwitchOn						: TIME;									//Delay befor the generator is switching on
	{attribute 'hide'}
	tTimDelayOutput						: TIME := T#5S;							//Delay Time to write some Data to the Output
	{attribute 'hide'}
	stSetupGenerator					: ST_Setup_Generator;					//Setup Generator
END_VAR
VAR_OUTPUT
	{attribute 'hide'}
	stDataGeneratorOut					: ST_Generator_Output;					//Generator Output data
	{attribute 'hide'}
	stDataGeneratorOutDelay				: ST_Generator_Output;					//Generator Output data with delay
END_VAR
VAR
	FPReset								: R_TRIG;								//Internal positive edge
	FPResetIntern						: R_TRIG;								//Internal positive edge
	FPEnable							: R_TRIG;								//Internal positive Edge
	FNEnable							: F_TRIG;								//Internal negative Edge
	timDelayOutputs						: TON;									//Timer to send Data with Delay to the outputs
	timGenEin							: TON;									//Timer to switch on the generator
	timResetOut							: TOF;									//Timer Reset Out
END_VAR

//Creator : Kai Ebensperger
//Company : Lynus AG
//Date : 28.05.2021
//Version : 1.0.0.0

//With this function its possible to control the basics from a generator
//The generator is switching on and off with the SOC from the battery

(*---------------------------------------------------------------Limit Inputs-------------------------------------------------------------------------------*)

dwBatterySOC := LIMIT(0,dwBatterySOC,100);

IF stSetupGenerator.byEnableSOC > stSetupGenerator.byDisableSOC THEN stSetupGenerator.byDisableSOC := stSetupGenerator.byEnableSOC + 1; END_IF

stSetupGenerator.byDisableSOC := LIMIT(1,stSetupGenerator.byDisableSOC,100);
	stSetupGenerator.byEnableSOC := LIMIT(0,stSetupGenerator.byEnableSOC,100);
		tDelaySwitchOn := LIMIT(T#10S,tDelaySwitchOn,T#2M);
		
IF IsFinite(F_LREAL(lrTotalCounterEnergy_Consumption)) THEN lrTotalCounterEnergy_Consumption := LIMIT(0,lrTotalCounterEnergy_Consumption,999999999999999); END_IF
	IF IsFinite(F_LREAL(lrTotalCounterEnergy_Production)) THEN lrTotalCounterEnergy_Production := LIMIT(0,lrTotalCounterEnergy_Production,999999999999999); END_IF
		IF IsFinite(F_LREAL(lrCounterEnergyT1_Consumption)) THEN lrCounterEnergyT1_Consumption := LIMIT(0,lrCounterEnergyT1_Consumption,999999999999999); END_IF
			IF IsFinite(F_LREAL(lrCounterEnergyT2_Consumption)) THEN lrCounterEnergyT2_Consumption := LIMIT(0,lrCounterEnergyT2_Consumption,999999999999999); END_IF
				IF IsFinite(F_LREAL(lrCounterEnergyT1_Production)) THEN lrCounterEnergyT1_Production := LIMIT(0,lrCounterEnergyT1_Production,999999999999999); END_IF
					IF IsFinite(F_LREAL(lrCounterEnergyT2_Production)) THEN lrCounterEnergyT2_Production := LIMIT(0,lrCounterEnergyT2_Production,999999999999999); END_IF
						lrPowerGenerator := LIMIT(-999999999999999,lrPowerGenerator,999999999999999);
	
(*---------------------------------------------------------------------------enable----------------------------------------------------------------------------------*)

stDataGeneratorOut.bEnabled := bEnable;

(*-----------------------------------------------------------------------------Error-Warning and Reset----------------------------------------------------------------------------*)

IF bWarning THEN stDataGeneratorOut.byErrorWarning := 1; END_IF 
	IF bError THEN stDataGeneratorOut.byErrorWarning := 2; END_IF

FPReset(CLK:= stSetupGenerator.bReset AND stDataGeneratorOut.byErrorWarning <> 0, Q=> ); 

timResetOut(IN:= FPReset.Q, PT:= T#2S, Q=> , ET=> );	

	stDataGeneratorOut.bSReset := timResetOut.Q;

FPResetIntern(CLK:= bReset, Q=> );	
	
IF NOT bError AND NOT bWarning AND FPResetIntern.Q THEN stDataGeneratorOut.byErrorWarning := 0; END_IF

//Messages and Error Codes
IF stDataGeneratorOut.byErrorWarning = 1 AND iWarningCode = 0 THEN stDataGeneratorOut.eMessage := E_Message_Generator.eNoConnectionToBackend;
ELSIF stDataGeneratorOut.byErrorWarning = 2 AND iErrorCode = 0 THEN stDataGeneratorOut.eMessage := E_Message_Generator.eGeneratorError;
ELSIF stDataGeneratorOut.byErrorWarning = 2 AND iErrorCode = 1 THEN stDataGeneratorOut.eMessage := E_Message_Generator.eTooMuchGenerators;
ELSE stDataGeneratorOut.eMessage := E_Message_Generator.eNoMessage; 
END_IF

(*----------------------------------------------------------------------------Logic------------------------------------------------------------------------------------*)

//Switch on
timGenEin(IN:= bEnable AND stDataGeneratorOut.byErrorWarning <> 2 AND dwBatterySOC <= stSetupGenerator.byEnableSOC, PT:= tDelaySwitchOn, Q=> , ET=> );
IF timGenEin.Q THEN stDataGeneratorOut.bOutput := TRUE; END_IF 

//Switch off
IF NOT bEnable OR stDataGeneratorOut.byErrorWarning = 2 OR dwBatterySOC >= stSetupGenerator.byDisableSOC THEN stDataGeneratorOut.bOutput := FALSE; END_IF 

(*------------------------------------------------------------------Power Data----------------------------------------------------------------------------------------------*)

timDelayOutputs(IN:= bWriteWithDelay AND bEnable AND NOT timDelayOutputs.Q, PT:= tTimDelayOutput, Q=> , ET=> );
	FPEnable(CLK:= bEnable, Q=> );
		FNEnable(CLK:= bEnable, Q=> );

IF bEnable THEN
	stDataGeneratorOut.lrPower:= LINT_TO_LREAL(LREAL_TO_LINT((lrPowerGenerator / 1000) * 100)) / 100;
		IF IsFinite(F_LREAL(lrCounterEnergyT1_Consumption)) THEN stDataGeneratorOut.lrCounterEnergyT1_Consumption := LINT_TO_LREAL(LREAL_TO_LINT((lrCounterEnergyT1_Consumption / 1000) * 100)) / 100; END_IF
			IF IsFinite(F_LREAL(lrCounterEnergyT2_Consumption)) THEN stDataGeneratorOut.lrCounterEnergyT2_Consumption := LINT_TO_LREAL(LREAL_TO_LINT((lrCounterEnergyT2_Consumption / 1000) * 100)) / 100; END_IF
				IF IsFinite(F_LREAL(lrCounterEnergyT1_Production)) THEN stDataGeneratorOut.lrCounterEnergyT1_Production := LINT_TO_LREAL(LREAL_TO_LINT((lrCounterEnergyT1_Production / 1000) * 100)) / 100; END_IF
					IF IsFinite(F_LREAL(lrCounterEnergyT2_Production)) THEN stDataGeneratorOut.lrCounterEnergyT2_Production := LINT_TO_LREAL(LREAL_TO_LINT((lrCounterEnergyT2_Production / 1000) * 100)) / 100; END_IF
						IF IsFinite(F_LREAL(lrTotalCounterEnergy_Consumption)) THEN stDataGeneratorOut.lrTotalCounterEnergy_Consumption := LINT_TO_LREAL(LREAL_TO_LINT((lrTotalCounterEnergy_Consumption / 1000) * 100)) / 100; END_IF
							IF IsFinite(F_LREAL(lrTotalCounterEnergy_Production)) THEN stDataGeneratorOut.lrTotalCounterEnergy_Production := LINT_TO_LREAL(LREAL_TO_LINT((lrTotalCounterEnergy_Production / 1000) * 100)) / 100; END_IF 	
			
	IF stDataGeneratorOut.lrPower < 0 THEN
		stDataGeneratorOut.lrPowerProduction := 0;
		stDataGeneratorOut.lrPowerConsumption := (stDataGeneratorOut.lrPower * - 1);
	ELSIF stDataGeneratorOut.lrPower > 0 THEN
		stDataGeneratorOut.lrPowerProduction := stDataGeneratorOut.lrPower;
		stDataGeneratorOut.lrPowerConsumption := 0;
	ELSIF stDataGeneratorOut.lrPower = 0 THEN
		stDataGeneratorOut.lrPowerProduction := 0;
		stDataGeneratorOut.lrPowerConsumption := 0;
	END_IF
ELSE	
	stDataGeneratorOut.lrPower := 0;
		stDataGeneratorOut.lrCounterEnergyT1_Consumption := 0;
			stDataGeneratorOut.lrCounterEnergyT2_Consumption := 0;
				stDataGeneratorOut.lrCounterEnergyT1_Production := 0;
					stDataGeneratorOut.lrCounterEnergyT2_Production := 0;
						stDataGeneratorOut.lrPowerProduction := 0;
							stDataGeneratorOut.lrPowerConsumption := 0;	
								stDataGeneratorOut.lrTotalCounterEnergy_Consumption := 0;
									stDataGeneratorOut.lrTotalCounterEnergy_Production := 0;
END_IF

(*---------------------------------------------------------------Outputs-------------------------------------------------------------------------------*)

//Write with Delay or without
IF (bWriteWithDelay AND (timDelayOutputs.Q OR FPEnable.Q OR FNEnable.Q)) OR NOT bWriteWithDelay THEN
	stDataGeneratorOutDelay := stDataGeneratorOut; 
END_IF

END_FUNCTION_BLOCK

// ---- Energy/FBs Internal/Grid/FB_GridConnection.TcPOU
{attribute 'hide_all_locals'}
{attribute 'conditionalshow'}
FUNCTION_BLOCK FB_GridConnection
VAR_INPUT
	{attribute 'hide'}
	bEnable								: BOOL;						//Enable or disable the function
	{attribute 'hide'}
	bError								: BOOL;						//Grid Error
	{attribute 'hide'}
	bWarning							: BOOL;						//Grid Warning
	{attribute 'hide'}
	bWriteWithDelay						: BOOL;						//Write with Delay the Data to the output (Not al Output Data is writen with Delay)
	{attribute 'hide'}
	iErrorCode							: INT;						//Error Code from external Grid
	{attribute 'hide'}
	iWarningCode						: INT;						//Warning Code from external Grid
	{attribute 'hide'}
	lrTotalCounterEnergy_Consumption	: LREAL;					//Total Counter for Energy consumption with unit Wh
	{attribute 'hide'}
	lrTotalCounterEnergy_Production		: LREAL;					//Total Counter for Energy production with unit Wh
	{attribute 'hide'}
	lrCounterEnergyT1_Consumption		: LREAL;					//Total counter for energy Tariff 1 consumption with unit Wh
	{attribute 'hide'}
	lrCounterEnergyT2_Consumption		: LREAL;					//Total counter for energy Tariff 2 consumption with unit Wh
	{attribute 'hide'}
	lrCounterEnergyT1_Production		: LREAL;					//Total counter for energy Tariff 1 production with unit Wh
	{attribute 'hide'}
	lrCounterEnergyT2_Production		: LREAL;					//Total counter for energy Tariff 2 production with unit Wh
	{attribute 'hide'}
	lrPowerGrid							: LREAL;					//Input Value from the power of the Grid with unit W
	{attribute 'hide'}
	rSizeGridConn						: REAL;						//Max size from the grid connection with unit KW
	{attribute 'hide'}
	tTimDelayOutput						: TIME := T#5S;				//Delay Time to write some Data to the Output
END_VAR
VAR_OUTPUT
	{attribute 'hide'}
	stDataGridOut						: ST_GridConnection_Output;	//Grid output data	
	{attribute 'hide'}
	stDataGridOutDelay					: ST_GridConnection_Output;	//Grid output data with delay	
END_VAR
VAR
	FPEnable							: R_TRIG;					//Internal positive Edge
	FNEnable							: F_TRIG;					//Internal negative Edge
	timDelayOutputs						: TON;						//Timer to send Data with Delay to the outputs
END_VAR

//Creator : Kai Ebensperger
//Company : Lynus AG
//Date : 28.05.2021
//Version : 1.0.0.0

//With this function its possible to handle the general data from a grid connection

(*---------------------------------------------------------------Check the limits of the inputs-------------------------------------------------------------------------------*)

rSizeGridConn := LIMIT(0,rSizeGridConn,2000);

IF IsFinite(F_LREAL(lrTotalCounterEnergy_Consumption)) THEN lrTotalCounterEnergy_Consumption := LIMIT(0,lrTotalCounterEnergy_Consumption,999999999999999); END_IF
	IF IsFinite(F_LREAL(lrTotalCounterEnergy_Production)) THEN lrTotalCounterEnergy_Production := LIMIT(0,lrTotalCounterEnergy_Production,999999999999999); END_IF
		IF IsFinite(F_LREAL(lrCounterEnergyT1_Consumption)) THEN lrCounterEnergyT1_Consumption := LIMIT(0,lrCounterEnergyT1_Consumption,999999999999999); END_IF
			IF IsFinite(F_LREAL(lrCounterEnergyT2_Consumption)) THEN lrCounterEnergyT2_Consumption := LIMIT(0,lrCounterEnergyT2_Consumption,999999999999999); END_IF
				IF IsFinite(F_LREAL(lrCounterEnergyT1_Production)) THEN lrCounterEnergyT1_Production := LIMIT(0,lrCounterEnergyT1_Production,999999999999999); END_IF
					IF IsFinite(F_LREAL(lrCounterEnergyT2_Production)) THEN lrCounterEnergyT2_Production := LIMIT(0,lrCounterEnergyT2_Production,999999999999999); END_IF
						lrPowerGrid := LIMIT(-999999999999999,lrPowerGrid,999999999999999);

(*---------------------------------------------------------------------------Enable----------------------------------------------------------------------------------*)

stDataGridOut.bEnabled := bEnable;

(*------------------------------------------------------------------Power data----------------------------------------------------------------------------------------------*)
stDataGridOut.rSizeGridConn := DINT_TO_REAL(REAL_TO_DINT((rSizeGridConn) * 100)) / 100;

timDelayOutputs(IN:= bWriteWithDelay AND bEnable AND NOT timDelayOutputs.Q, PT:= tTimDelayOutput, Q=> , ET=> );
	FPEnable(CLK:= bEnable, Q=> );
		FNEnable(CLK:= bEnable, Q=> );

IF bEnable THEN
	stDataGridOut.lrPower:= LINT_TO_LREAL(LREAL_TO_LINT((lrPowerGrid / 1000) * 100)) / 100;
		IF IsFinite(F_LREAL(lrCounterEnergyT1_Consumption)) THEN stDataGridOut.lrCounterEnergyT1_Consumption := LINT_TO_LREAL(LREAL_TO_LINT((lrCounterEnergyT1_Consumption / 1000) * 100)) / 100; END_IF
			IF IsFinite(F_LREAL(lrCounterEnergyT2_Consumption)) THEN stDataGridOut.lrCounterEnergyT2_Consumption := LINT_TO_LREAL(LREAL_TO_LINT((lrCounterEnergyT2_Consumption / 1000) * 100)) / 100; END_IF
				IF IsFinite(F_LREAL(lrCounterEnergyT1_Production)) THEN stDataGridOut.lrCounterEnergyT1_Production := LINT_TO_LREAL(LREAL_TO_LINT((lrCounterEnergyT1_Production / 1000) * 100)) / 100; END_IF
					IF IsFinite(F_LREAL(lrCounterEnergyT2_Production)) THEN stDataGridOut.lrCounterEnergyT2_Production := LINT_TO_LREAL(LREAL_TO_LINT((lrCounterEnergyT2_Production / 1000) * 100)) / 100; END_IF
						IF IsFinite(F_LREAL(lrTotalCounterEnergy_Consumption)) THEN stDataGridOut.lrTotalCounterEnergy_Consumption := LINT_TO_LREAL(LREAL_TO_LINT((lrTotalCounterEnergy_Consumption / 1000) * 100)) / 100; END_IF
							IF IsFinite(F_LREAL(lrTotalCounterEnergy_Production)) THEN stDataGridOut.lrTotalCounterEnergy_Production := LINT_TO_LREAL(LREAL_TO_LINT((lrTotalCounterEnergy_Production / 1000) * 100)) / 100; END_IF 
						
		IF stDataGridOut.lrPower < 0 THEN
				stDataGridOut.lrPowerProduction := (stDataGridOut.lrPower * - 1);
				stDataGridOut.lrPowerConsumption := 0;
		ELSIF stDataGridOut.lrPower > 0 THEN
				stDataGridOut.lrPowerProduction := 0;
				stDataGridOut.lrPowerConsumption := stDataGridOut.lrPower;
		ELSIF stDataGridOut.lrPower = 0 THEN
				stDataGridOut.lrPowerProduction := 0;
				stDataGridOut.lrPowerConsumption := 0;
		END_IF															
ELSE																	
	stDataGridOut.lrPower := 0;
		stDataGridOut.lrCounterEnergyT1_Consumption := 0;
			stDataGridOut.lrCounterEnergyT2_Consumption := 0;
				stDataGridOut.lrCounterEnergyT1_Production := 0;
					stDataGridOut.lrCounterEnergyT2_Production := 0;
						stDataGridOut.lrPowerProduction := 0;
							stDataGridOut.lrPowerConsumption := 0;
								stDataGridOut.lrTotalCounterEnergy_Consumption := 0;
									stDataGridOut.lrTotalCounterEnergy_Production := 0;
END_IF	

(*------------------------------------------------------------------Error and Warning----------------------------------------------------------------------------------------------*)

stDataGridOut.byErrorWarning := 0;
	IF bWarning THEN stDataGridOut.byErrorWarning := 1; END_IF 
	IF bError THEN stDataGridOut.byErrorWarning := 2; END_IF

//Messages and Error Codes
IF stDataGridOut.byErrorWarning = 1 AND iWarningCode = 0 THEN stDataGridOut.eMessage := E_Message_Grid.eNoConnectionToBackend;
ELSIF stDataGridOut.byErrorWarning = 2 AND iErrorCode = 0 THEN stDataGridOut.eMessage := E_Message_Grid.eGridError;
ELSIF stDataGridOut.byErrorWarning = 2 AND iErrorCode = 1 THEN stDataGridOut.eMessage := E_Message_Grid.eTooMuchGrids;
ELSE stDataGridOut.eMessage := E_Message_Grid.eNoMessage; 
END_IF

(*---------------------------------------------------------------Outputs-------------------------------------------------------------------------------*)

//Write with Delay or without
IF (bWriteWithDelay AND (timDelayOutputs.Q OR FPEnable.Q OR FNEnable.Q)) OR NOT bWriteWithDelay THEN
	stDataGridOutDelay := stDataGridOut; 
END_IF

END_FUNCTION_BLOCK

// ---- Energy/FBs Internal/Heating Pump/FB_HeatingPump.TcPOU
{attribute 'hide_all_locals'}
{attribute 'conditionalshow'}
FUNCTION_BLOCK FB_HeatingPump
VAR_INPUT
	{attribute 'hide'}
	bEnable								: BOOL;									//Enable or dissable the function
	{attribute 'hide'}
	bError								: BOOL;									//Error Heating pump
	{attribute 'hide'}
	bWarning							: BOOL;									//Warning Heating pump
	{attribute 'hide'}
	bIsStepSwitched						: BOOL;									//Heating pump is step switched or not
	{attribute 'hide'}
	bEPOIsActive						: BOOL;									//Emergency power operation is active
	{attribute 'hide'}
	bExternalLock						: BOOL;									//External lock (All functions are locked)
	{attribute 'hide'}
	bReset								: BOOL;									//Reset the Heating pup after an error with the output reset and a negative edge
	{attribute 'hide'}
	bExternalOnCommand					: BOOL;									//External On command to switch on the heating pump
	{attribute 'hide'}
	bWriteWithDelay						: BOOL;									//Write with Delay the Data to the output (Not al Output Data is writen with Delay)
	{attribute 'hide'}
	bHPIsRunning						: BOOL;									//Feedback from the Heating pump if he is running (Need for min run time)
	{attribute 'hide'}
	iErrorCode							: INT;									//Error Code from external HP
	{attribute 'hide'}
	iWarningCode						: INT;									//Warning Code from external HP
	{attribute 'hide'}
	dwBatterySOC						: DWORD;								//Actual Battery SOC in %
	{attribute 'hide'}
	diNumberOfHP						: DINT;									//Number of heating pump what is calculatet by a external function
	{attribute 'hide'}
	rBoilerTempHeatingSys				: REAL;									//Boilertemperatur Heating system with the unit °C
	{attribute 'hide'}
	rBoilerTempServiceWater				: REAL;									//Boilertemperatur Service water with the unit °C
	{attribute 'hide'}
	rFlowTemp							: REAL;									//Flow temperatur heating pump with the unit °C
	{attribute 'hide'}
	rReturnTemp							: REAL;									//Return temperatur heating pump with the unit °C
	{attribute 'hide'}
	rFlowTempEnergySource				: REAL;									//Flow temperatur energy source heating pump with the unit °C
	{attribute 'hide'}
	rReturnTempEnergySource				: REAL;									//Return temperatur energy source heating pump with the unit °C
	{attribute 'hide'}
	lrSizeGridConnection				: LREAL;								//Max size from the grid connection in kW
	{attribute 'hide'}
	lrGridPower							: LREAL;								//Actual Grid power in kW
	{attribute 'hide'}
	lrTotalCounterEnergy_Consumption	: LREAL;								//Total Counter for Energy consumption with unit Wh
	{attribute 'hide'}
	lrTotalCounterEnergy_Production		: LREAL;								//Total Counter for Energy production with unit Wh
	{attribute 'hide'}
	lrCounterEnergyT1_Consumption		: LREAL;								//Total counter for energy Tariff 1 consumption with unit Wh
	{attribute 'hide'}
	lrCounterEnergyT2_Consumption		: LREAL;								//Total counter for energy Tariff 2 consumption with unit Wh
	{attribute 'hide'}
	lrCounterEnergyT1_Production		: LREAL;								//Total counter for energy Tariff 1 production with unit Wh
	{attribute 'hide'}
	lrCounterEnergyT2_Production		: LREAL;								//Total counter for energy Tariff 2 production with unit Wh
	{attribute 'hide'}
	lrCounterThermalEnergy_Heating		: LREAL;								//Total Counter for thermal Energy from the heating system with unit Wh
	{attribute 'hide'}
	lrCounterThermalEnergy_Water		: LREAL;								//Total Counter for thermal Energy from the service water system with unit Wh
	{attribute 'hide'}
	lrElPowerHP							: LREAL;								//Input Value from the power of the Heating pump with unit W
	{attribute 'hide'}
	arrTargetPower						: ARRAY[1..2] OF REAL;					//Target power from 0% to +100% for each step (0% to 100%) 
	{attribute 'hide'}
	tOnDelayExternalOn					: TIME := T#2M;							//On delay before the pump is switching on with external on command
	{attribute 'hide'}
	tOffDelayExternalOn					: TIME := T#1H;							//Off delay when the pump was switching on with external on command
	{attribute 'hide'}
	tMinOnTime							: TIME := T#30M;						//Minimum On time for the HP in the surplus mode 
	{attribute 'hide'}
	tTimDelayOutput						: TIME := T#5S;							//Delay Time to write some Data to the Output
	{attribute 'hide'}	
	stSystemTime						: ST_Systemtime;						//Local system time
	{attribute 'hide'}
	stSetupHP							: ST_Setup_HP;							//Setup heating pump
END_VAR
VAR_OUTPUT
	{attribute 'hide'}
	stDataHPOut							: ST_HP_Output;							//Heating pump output data
	{attribute 'hide'}
	stDataHPOutDelay					: ST_HP_Output;							//Heating pump output data with delay
	{attribute 'hide'}
	arrPercentValuesSteps				: ARRAY[1..2] OF REAL;					//Percent values from the Steps
END_VAR
VAR
	FPTimeEn							: R_TRIG;								//Internal positive edge
	FPTimeDis							: R_TRIG;								//Internal positive edge
	FPReset								: R_TRIG;								//Internal positive edge
	FPResetIntern						: R_TRIG;								//Internal positive edge
	FPExternalOnCommand					: R_TRIG;								//Internal positive edge
	FPStartMinOnTimer					: R_TRIG;								//Internal postive edge
	FPEnable							: R_TRIG;								//Internal positive Edge
	FNEnable							: F_TRIG;								//Internal negative Edge
	timDelayOutputs						: TON;									//Timer to send Data with Delay to the outputs
	timResetOut							: TOF;									//Timer to reset the error
	timMinOnInStep4						: TOF;									//Timer for the minimum on time in the step 4 in the surplus mode.
	timOnDelayExternalOn				: TON;									//Timer to start the pump with a delay when external on command is active
	timOffDelayExternalOn				: TON;									//Timer to stop the pump with a delay after the pump was running in the external on command mode
	timSOCOff							: TON;									//Timer to dissable the Device when the SOC from the Battery is under the Setpoint
	bEnableTimeFunction					: BOOL;									//Enable the time function
	byLPMaxPower						: BYTE;									//Loop to limit the max power and the target power from the ems
	byLPNumberOfSteps					: BYTE;									//Loop to count the numbers of active steps
	byLPMaxPowerLimit					: BYTE;									//Loop to limit the max power at the output with 1 comma
	byLPCalcStepPower					: BYTE;									//Loop to calcualte the power from each step
	byLPCalcPercentPowerSteps			: BYTE;									//Loop to calcualte the % power from each step
	byLPMaxIsReached					: BYTE;									//Loop to check if each step has reached the maximum of target power or not
	iStateIntStep3						: INT;									//Internal state machine in general step 3
	uiState								: UINT;									//State Maschine
	rSumOfSteps							: REAL;									//Total sum of each steps in kW
	arrMaxPower							: ARRAY[1..2] OF REAL; 					//Maximum power of the consumer in kW (Per stage) [1] = Increased operation [2] = Maximum operation
	arrMaxIsReached						: ARRAY[1..2] OF BOOL;					//Array in wich is saved when the target power from each step is >= 100%
END_VAR

//Creator : Kai Ebensperger
//Company : Lynus AG
//Date : 28.05.2021
//Version : 1.0.0.0

